// TIA Portal project "modbus-tcp-as-server" (V17)

(* hardware
DEVICE "S7-1200 station_1"  S7-1200 Station
   slot 0: "Rack_0"  S7-1200 Rack  Rack  V1.0
   slot 1: "PLC_1"  CPU 1214C DC/DC/DC  6ES7 214-1AG40-0XB0  V4.5
   slot 101: "CM 1241 (RS422/485)_1"  6ES7 241-1CH32-0XB0  V2.2
*)

// ===== PLC "PLC_1"  CPU 1214C DC/DC/DC =====

VAR_GLOBAL   // PLC tag table "Default tag table"
   "System_Byte" AT %MB1 : Byte;
   "FirstScan" AT %M1.0 : Bool;
   "DiagStatusUpdate" AT %M1.1 : Bool;
   "AlwaysTRUE" AT %M1.2 : Bool;
   "AlwaysFALSE" AT %M1.3 : Bool;
   "Clock_Byte" AT %MB0 : Byte;
   "Clock_10Hz" AT %M0.0 : Bool;
   "Clock_5Hz" AT %M0.1 : Bool;
   "Clock_2.5Hz" AT %M0.2 : Bool;
   "Clock_2Hz" AT %M0.3 : Bool;
   "Clock_1.25Hz" AT %M0.4 : Bool;
   "Clock_1Hz" AT %M0.5 : Bool;
   "Clock_0.625Hz" AT %M0.6 : Bool;
   "Clock_0.5Hz" AT %M0.7 : Bool;
   "Bit1s" AT %M2.0 : Bool;
END_VAR

// folder: Global

DATA_BLOCK "ConfigModel"   // DB1
{ S7_Optimized_Access := 'TRUE' }
VERSION : 0.1
   VAR
      Info : Struct
         ProjectName : String := 'Modbus Tcp As Server';
         Client : String := 'Than Ho';
         Authour : String := 'thanho.dut@gmail.com';
         Tel : String := '0933600195';
         "Version" : String := '2023.05.23.001';
      END_STRUCT;
   END_VAR
BEGIN
END_DATA_BLOCK

DATA_BLOCK "ModbusModel"   // DB3
{ S7_Optimized_Access := 'TRUE' }
VERSION : 0.1
   VAR
      Disconnect : Bool := FALSE;
      NDR : Bool := FALSE;   // Write data completed withou error
      DR : Bool := FALSE;   // Read data completed withou error
      Error : Bool := FALSE;   // Instruction finished with error
      Status : Word := 16#7006;   // Detailed error information
      Connect : TCON_IP_v4;
      HoldingRegisters : Array[0..4999] of Word;   // Data buffer write/read
   END_VAR
BEGIN
   Connect.InterfaceId := 64;
   Connect.ID := 16#0001;
   Connect.RemoteAddress.ADDR[1] := 16#00;
   Connect.RemoteAddress.ADDR[2] := 16#00;
   Connect.RemoteAddress.ADDR[3] := 16#00;
   Connect.RemoteAddress.ADDR[4] := 16#00;
   Connect.LocalPort := 502;
   Connect.ConnectionType := 16#0B;
   Connect.ActiveEstablished := FALSE;
   Connect.RemotePort := 0;
   HoldingRegisters[0] := 16#0000;
   HoldingRegisters[1] := 16#0000;
   HoldingRegisters[2] := 16#0000;
   HoldingRegisters[3] := 16#0000;
   HoldingRegisters[4] := 16#0000;
   HoldingRegisters[5] := 16#0000;
   HoldingRegisters[6] := 16#0000;
   HoldingRegisters[7] := 16#0000;
   HoldingRegisters[8] := 16#0000;
   HoldingRegisters[9] := 16#0000;
   HoldingRegisters[10] := 16#0000;
   HoldingRegisters[11] := 16#0000;
   HoldingRegisters[12] := 16#0000;
   HoldingRegisters[13] := 16#0000;
   HoldingRegisters[14] := 16#0000;
   HoldingRegisters[15] := 16#0000;
   HoldingRegisters[16] := 16#0000;
   HoldingRegisters[17] := 16#0000;
   HoldingRegisters[18] := 16#0000;
   HoldingRegisters[19] := 16#0000;
   HoldingRegisters[20] := 16#0000;
   HoldingRegisters[21] := 16#0000;
   HoldingRegisters[22] := 16#0000;
   HoldingRegisters[23] := 16#0000;
   HoldingRegisters[24] := 16#0000;
   HoldingRegisters[25] := 16#0000;
   HoldingRegisters[26] := 16#0000;
   HoldingRegisters[27] := 16#0000;
   HoldingRegisters[28] := 16#0000;
   HoldingRegisters[29] := 16#0000;
   HoldingRegisters[30] := 16#0000;
   HoldingRegisters[31] := 16#0000;
   HoldingRegisters[32] := 16#0000;
   HoldingRegisters[33] := 16#0000;
   HoldingRegisters[34] := 16#0000;
   HoldingRegisters[35] := 16#0000;
   HoldingRegisters[36] := 16#0000;
   HoldingRegisters[37] := 16#0000;
   HoldingRegisters[38] := 16#0000;
   HoldingRegisters[39] := 16#0000;
   HoldingRegisters[40] := 16#0000;
   HoldingRegisters[41] := 16#0000;
   HoldingRegisters[42] := 16#0000;
   HoldingRegisters[43] := 16#0000;
   HoldingRegisters[44] := 16#0000;
   HoldingRegisters[45] := 16#0000;
   HoldingRegisters[46] := 16#0000;
   HoldingRegisters[47] := 16#0000;
   HoldingRegisters[48] := 16#0000;
   HoldingRegisters[49] := 16#0000;
   HoldingRegisters[50] := 16#0000;
   HoldingRegisters[51] := 16#0000;
   HoldingRegisters[52] := 16#0000;
   HoldingRegisters[53] := 16#0000;
   HoldingRegisters[54] := 16#0000;
   HoldingRegisters[55] := 16#0000;
   HoldingRegisters[56] := 16#0000;
   HoldingRegisters[57] := 16#0000;
   HoldingRegisters[58] := 16#0000;
   HoldingRegisters[59] := 16#0000;
   HoldingRegisters[60] := 16#0000;
   HoldingRegisters[61] := 16#0000;
   HoldingRegisters[62] := 16#0000;
   HoldingRegisters[63] := 16#0000;
   HoldingRegisters[64] := 16#0000;
   HoldingRegisters[65] := 16#0000;
   HoldingRegisters[66] := 16#0000;
   HoldingRegisters[67] := 16#0000;
   HoldingRegisters[68] := 16#0000;
   HoldingRegisters[69] := 16#0000;
   HoldingRegisters[70] := 16#0000;
   HoldingRegisters[71] := 16#0000;
   HoldingRegisters[72] := 16#0000;
   HoldingRegisters[73] := 16#0000;
   HoldingRegisters[74] := 16#0000;
   HoldingRegisters[75] := 16#0000;
   HoldingRegisters[76] := 16#0000;
   HoldingRegisters[77] := 16#0000;
   HoldingRegisters[78] := 16#0000;
   HoldingRegisters[79] := 16#0000;
   HoldingRegisters[80] := 16#0000;
   HoldingRegisters[81] := 16#0000;
   HoldingRegisters[82] := 16#0000;
   HoldingRegisters[83] := 16#0000;
   HoldingRegisters[84] := 16#0000;
   HoldingRegisters[85] := 16#0000;
   HoldingRegisters[86] := 16#0000;
   HoldingRegisters[87] := 16#0000;
   HoldingRegisters[88] := 16#0000;
   HoldingRegisters[89] := 16#0000;
   HoldingRegisters[90] := 16#0000;
   HoldingRegisters[91] := 16#0000;
   HoldingRegisters[92] := 16#0000;
   HoldingRegisters[93] := 16#0000;
   HoldingRegisters[94] := 16#0000;
   HoldingRegisters[95] := 16#0000;
   HoldingRegisters[96] := 16#0000;
   HoldingRegisters[97] := 16#0000;
   HoldingRegisters[98] := 16#0000;
   HoldingRegisters[99] := 16#0000;
   HoldingRegisters[100] := 16#0006;
   HoldingRegisters[101] := 16#0000;
   HoldingRegisters[102] := 16#0000;
   HoldingRegisters[103] := 16#0000;
   HoldingRegisters[104] := 16#0000;
   HoldingRegisters[105] := 16#0000;
   HoldingRegisters[106] := 16#0000;
   HoldingRegisters[107] := 16#0000;
   HoldingRegisters[108] := 16#0000;
   HoldingRegisters[109] := 16#0000;
   HoldingRegisters[110] := 16#0000;
   HoldingRegisters[111] := 16#0000;
   HoldingRegisters[112] := 16#0000;
   HoldingRegisters[113] := 16#0000;
   HoldingRegisters[114] := 16#0000;
   HoldingRegisters[115] := 16#0000;
   HoldingRegisters[116] := 16#0000;
   HoldingRegisters[117] := 16#0000;
   HoldingRegisters[118] := 16#0000;
   HoldingRegisters[119] := 16#0000;
   HoldingRegisters[120] := 16#0000;
   HoldingRegisters[121] := 16#0000;
   HoldingRegisters[122] := 16#0000;
   HoldingRegisters[123] := 16#0000;
   HoldingRegisters[124] := 16#0000;
   HoldingRegisters[125] := 16#0000;
   HoldingRegisters[126] := 16#0000;
   HoldingRegisters[127] := 16#0000;
   HoldingRegisters[128] := 16#0000;
   HoldingRegisters[129] := 16#0000;
   HoldingRegisters[130] := 16#0000;
   HoldingRegisters[131] := 16#0000;
   HoldingRegisters[132] := 16#0000;
   HoldingRegisters[133] := 16#0000;
   HoldingRegisters[134] := 16#0000;
   HoldingRegisters[135] := 16#0000;
   HoldingRegisters[136] := 16#0000;
   HoldingRegisters[137] := 16#0000;
   HoldingRegisters[138] := 16#0000;
   HoldingRegisters[139] := 16#0000;
   HoldingRegisters[140] := 16#0000;
   HoldingRegisters[141] := 16#0000;
   HoldingRegisters[142] := 16#0000;
   HoldingRegisters[143] := 16#0000;
   HoldingRegisters[144] := 16#0000;
   HoldingRegisters[145] := 16#0000;
   HoldingRegisters[146] := 16#0000;
   HoldingRegisters[147] := 16#0000;
   HoldingRegisters[148] := 16#0000;
   HoldingRegisters[149] := 16#0000;
   HoldingRegisters[150] := 16#0000;
   HoldingRegisters[151] := 16#0000;
   HoldingRegisters[152] := 16#0000;
   HoldingRegisters[153] := 16#0000;
   HoldingRegisters[154] := 16#0000;
   HoldingRegisters[155] := 16#0000;
   HoldingRegisters[156] := 16#0000;
   HoldingRegisters[157] := 16#0000;
   HoldingRegisters[158] := 16#0000;
   HoldingRegisters[159] := 16#0000;
   HoldingRegisters[160] := 16#0000;
   HoldingRegisters[161] := 16#0000;
   HoldingRegisters[162] := 16#0000;
   HoldingRegisters[163] := 16#0000;
   HoldingRegisters[164] := 16#0000;
   HoldingRegisters[165] := 16#0000;
   HoldingRegisters[166] := 16#0000;
   HoldingRegisters[167] := 16#0000;
   HoldingRegisters[168] := 16#0000;
   HoldingRegisters[169] := 16#0000;
   HoldingRegisters[170] := 16#0000;
   HoldingRegisters[171] := 16#0000;
   HoldingRegisters[172] := 16#0000;
   HoldingRegisters[173] := 16#0000;
   HoldingRegisters[174] := 16#0000;
   HoldingRegisters[175] := 16#0000;
   HoldingRegisters[176] := 16#0000;
   HoldingRegisters[177] := 16#0000;
   HoldingRegisters[178] := 16#0000;
   HoldingRegisters[179] := 16#0000;
   HoldingRegisters[180] := 16#0000;
   HoldingRegisters[181] := 16#0000;
   HoldingRegisters[182] := 16#0000;
   HoldingRegisters[183] := 16#0000;
   HoldingRegisters[184] := 16#0000;
   HoldingRegisters[185] := 16#0000;
   HoldingRegisters[186] := 16#0000;
   HoldingRegisters[187] := 16#0000;
   HoldingRegisters[188] := 16#0000;
   HoldingRegisters[189] := 16#0000;
   HoldingRegisters[190] := 16#0000;
   HoldingRegisters[191] := 16#0000;
   HoldingRegisters[192] := 16#0000;
   HoldingRegisters[193] := 16#0000;
   HoldingRegisters[194] := 16#0000;
   HoldingRegisters[195] := 16#0000;
   HoldingRegisters[196] := 16#0000;
   HoldingRegisters[197] := 16#0000;
   HoldingRegisters[198] := 16#0000;
   HoldingRegisters[199] := 16#0000;
   HoldingRegisters[200] := 16#0000;
   HoldingRegisters[201] := 16#0000;
   HoldingRegisters[202] := 16#0000;
   HoldingRegisters[203] := 16#0000;
   HoldingRegisters[204] := 16#0000;
   HoldingRegisters[205] := 16#0000;
   HoldingRegisters[206] := 16#0000;
   HoldingRegisters[207] := 16#0000;
   HoldingRegisters[208] := 16#0000;
   HoldingRegisters[209] := 16#0000;
   HoldingRegisters[210] := 16#0000;
   HoldingRegisters[211] := 16#0000;
   HoldingRegisters[212] := 16#0000;
   HoldingRegisters[213] := 16#0000;
   HoldingRegisters[214] := 16#0000;
   HoldingRegisters[215] := 16#0000;
   HoldingRegisters[216] := 16#0000;
   HoldingRegisters[217] := 16#0000;
   HoldingRegisters[218] := 16#0000;
   HoldingRegisters[219] := 16#0000;
   HoldingRegisters[220] := 16#0000;
   HoldingRegisters[221] := 16#0000;
   HoldingRegisters[222] := 16#0000;
   HoldingRegisters[223] := 16#0000;
   HoldingRegisters[224] := 16#0000;
   HoldingRegisters[225] := 16#0000;
   HoldingRegisters[226] := 16#0000;
   HoldingRegisters[227] := 16#0000;
   HoldingRegisters[228] := 16#0000;
   HoldingRegisters[229] := 16#0000;
   HoldingRegisters[230] := 16#0000;
   HoldingRegisters[231] := 16#0000;
   HoldingRegisters[232] := 16#0000;
   HoldingRegisters[233] := 16#0000;
   HoldingRegisters[234] := 16#0000;
   HoldingRegisters[235] := 16#0000;
   HoldingRegisters[236] := 16#0000;
   HoldingRegisters[237] := 16#0000;
   HoldingRegisters[238] := 16#0000;
   HoldingRegisters[239] := 16#0000;
   HoldingRegisters[240] := 16#0000;
   HoldingRegisters[241] := 16#0000;
   HoldingRegisters[242] := 16#0000;
   HoldingRegisters[243] := 16#0000;
   HoldingRegisters[244] := 16#0000;
   HoldingRegisters[245] := 16#0000;
   HoldingRegisters[246] := 16#0000;
   HoldingRegisters[247] := 16#0000;
   HoldingRegisters[248] := 16#0000;
   HoldingRegisters[249] := 16#0000;
   HoldingRegisters[250] := 16#0000;
   HoldingRegisters[251] := 16#0000;
   HoldingRegisters[252] := 16#0000;
   HoldingRegisters[253] := 16#0000;
   HoldingRegisters[254] := 16#0000;
   HoldingRegisters[255] := 16#0000;
   HoldingRegisters[256] := 16#0000;
   HoldingRegisters[257] := 16#0000;
   HoldingRegisters[258] := 16#0000;
   HoldingRegisters[259] := 16#0000;
   HoldingRegisters[260] := 16#0000;
   HoldingRegisters[261] := 16#0000;
   HoldingRegisters[262] := 16#0000;
   HoldingRegisters[263] := 16#0000;
   HoldingRegisters[264] := 16#0000;
   HoldingRegisters[265] := 16#0000;
   HoldingRegisters[266] := 16#0000;
   HoldingRegisters[267] := 16#0000;
   HoldingRegisters[268] := 16#0000;
   HoldingRegisters[269] := 16#0000;
   HoldingRegisters[270] := 16#0000;
   HoldingRegisters[271] := 16#0000;
   HoldingRegisters[272] := 16#0000;
   HoldingRegisters[273] := 16#0000;
   HoldingRegisters[274] := 16#0000;
   HoldingRegisters[275] := 16#0000;
   HoldingRegisters[276] := 16#0000;
   HoldingRegisters[277] := 16#0000;
   HoldingRegisters[278] := 16#0000;
   HoldingRegisters[279] := 16#0000;
   HoldingRegisters[280] := 16#0000;
   HoldingRegisters[281] := 16#0000;
   HoldingRegisters[282] := 16#0000;
   HoldingRegisters[283] := 16#0000;
   HoldingRegisters[284] := 16#0000;
   HoldingRegisters[285] := 16#0000;
   HoldingRegisters[286] := 16#0000;
   HoldingRegisters[287] := 16#0000;
   HoldingRegisters[288] := 16#0000;
   HoldingRegisters[289] := 16#0000;
   HoldingRegisters[290] := 16#0000;
   HoldingRegisters[291] := 16#0000;
   HoldingRegisters[292] := 16#0000;
   HoldingRegisters[293] := 16#0000;
   HoldingRegisters[294] := 16#0000;
   HoldingRegisters[295] := 16#0000;
   HoldingRegisters[296] := 16#0000;
   HoldingRegisters[297] := 16#0000;
   HoldingRegisters[298] := 16#0000;
   HoldingRegisters[299] := 16#0000;
   HoldingRegisters[300] := 16#0000;
   HoldingRegisters[301] := 16#0000;
   HoldingRegisters[302] := 16#0000;
   HoldingRegisters[303] := 16#0000;
   HoldingRegisters[304] := 16#0000;
   HoldingRegisters[305] := 16#0000;
   HoldingRegisters[306] := 16#0000;
   HoldingRegisters[307] := 16#0000;
   HoldingRegisters[308] := 16#0000;
   HoldingRegisters[309] := 16#0000;
   HoldingRegisters[310] := 16#0000;
   HoldingRegisters[311] := 16#0000;
   HoldingRegisters[312] := 16#0000;
   HoldingRegisters[313] := 16#0000;
   HoldingRegisters[314] := 16#0000;
   HoldingRegisters[315] := 16#0000;
   HoldingRegisters[316] := 16#0000;
   HoldingRegisters[317] := 16#0000;
   HoldingRegisters[318] := 16#0000;
   HoldingRegisters[319] := 16#0000;
   HoldingRegisters[320] := 16#0000;
   HoldingRegisters[321] := 16#0000;
   HoldingRegisters[322] := 16#0000;
   HoldingRegisters[323] := 16#0000;
   HoldingRegisters[324] := 16#0000;
   HoldingRegisters[325] := 16#0000;
   HoldingRegisters[326] := 16#0000;
   HoldingRegisters[327] := 16#0000;
   HoldingRegisters[328] := 16#0000;
   HoldingRegisters[329] := 16#0000;
   HoldingRegisters[330] := 16#0000;
   HoldingRegisters[331] := 16#0000;
   HoldingRegisters[332] := 16#0000;
   HoldingRegisters[333] := 16#0000;
   HoldingRegisters[334] := 16#0000;
   HoldingRegisters[335] := 16#0000;
   HoldingRegisters[336] := 16#0000;
   HoldingRegisters[337] := 16#0000;
   HoldingRegisters[338] := 16#0000;
   HoldingRegisters[339] := 16#0000;
   HoldingRegisters[340] := 16#0000;
   HoldingRegisters[341] := 16#0000;
   HoldingRegisters[342] := 16#0000;
   HoldingRegisters[343] := 16#0000;
   HoldingRegisters[344] := 16#0000;
   HoldingRegisters[345] := 16#0000;
   HoldingRegisters[346] := 16#0000;
   HoldingRegisters[347] := 16#0000;
   HoldingRegisters[348] := 16#0000;
   HoldingRegisters[349] := 16#0000;
   HoldingRegisters[350] := 16#0000;
   HoldingRegisters[351] := 16#0000;
   HoldingRegisters[352] := 16#0000;
   HoldingRegisters[353] := 16#0000;
   HoldingRegisters[354] := 16#0000;
   HoldingRegisters[355] := 16#0000;
   HoldingRegisters[356] := 16#0000;
   HoldingRegisters[357] := 16#0000;
   HoldingRegisters[358] := 16#0000;
   HoldingRegisters[359] := 16#0000;
   HoldingRegisters[360] := 16#0000;
   HoldingRegisters[361] := 16#0000;
   HoldingRegisters[362] := 16#0000;
   HoldingRegisters[363] := 16#0000;
   HoldingRegisters[364] := 16#0000;
   HoldingRegisters[365] := 16#0000;
   HoldingRegisters[366] := 16#0000;
   HoldingRegisters[367] := 16#0000;
   HoldingRegisters[368] := 16#0000;
   HoldingRegisters[369] := 16#0000;
   HoldingRegisters[370] := 16#0000;
   HoldingRegisters[371] := 16#0000;
   HoldingRegisters[372] := 16#0000;
   HoldingRegisters[373] := 16#0000;
   HoldingRegisters[374] := 16#0000;
   HoldingRegisters[375] := 16#0000;
   HoldingRegisters[376] := 16#0000;
   HoldingRegisters[377] := 16#0000;
   HoldingRegisters[378] := 16#0000;
   HoldingRegisters[379] := 16#0000;
   HoldingRegisters[380] := 16#0000;
   HoldingRegisters[381] := 16#0000;
   HoldingRegisters[382] := 16#0000;
   HoldingRegisters[383] := 16#0000;
   HoldingRegisters[384] := 16#0000;
   HoldingRegisters[385] := 16#0000;
   HoldingRegisters[386] := 16#0000;
   HoldingRegisters[387] := 16#0000;
   HoldingRegisters[388] := 16#0000;
   HoldingRegisters[389] := 16#0000;
   HoldingRegisters[390] := 16#0000;
   HoldingRegisters[391] := 16#0000;
   HoldingRegisters[392] := 16#0000;
   HoldingRegisters[393] := 16#0000;
   HoldingRegisters[394] := 16#0000;
   HoldingRegisters[395] := 16#0000;
   HoldingRegisters[396] := 16#0000;
   HoldingRegisters[397] := 16#0000;
   HoldingRegisters[398] := 16#0000;
   HoldingRegisters[399] := 16#0000;
   HoldingRegisters[400] := 16#0000;
   HoldingRegisters[401] := 16#0000;
   HoldingRegisters[402] := 16#0000;
   HoldingRegisters[403] := 16#0000;
   HoldingRegisters[404] := 16#0000;
   HoldingRegisters[405] := 16#0000;
   HoldingRegisters[406] := 16#0000;
   HoldingRegisters[407] := 16#0000;
   HoldingRegisters[408] := 16#0000;
   HoldingRegisters[409] := 16#0000;
   HoldingRegisters[410] := 16#0000;
   HoldingRegisters[411] := 16#0000;
   HoldingRegisters[412] := 16#0000;
   HoldingRegisters[413] := 16#0000;
   HoldingRegisters[414] := 16#0000;
   HoldingRegisters[415] := 16#0000;
   HoldingRegisters[416] := 16#0000;
   HoldingRegisters[417] := 16#0000;
   HoldingRegisters[418] := 16#0000;
   HoldingRegisters[419] := 16#0000;
   HoldingRegisters[420] := 16#0000;
   HoldingRegisters[421] := 16#0000;
   HoldingRegisters[422] := 16#0000;
   HoldingRegisters[423] := 16#0000;
   HoldingRegisters[424] := 16#0000;
   HoldingRegisters[425] := 16#0000;
   HoldingRegisters[426] := 16#0000;
   HoldingRegisters[427] := 16#0000;
   HoldingRegisters[428] := 16#0000;
   HoldingRegisters[429] := 16#0000;
   HoldingRegisters[430] := 16#0000;
   HoldingRegisters[431] := 16#0000;
   HoldingRegisters[432] := 16#0000;
   HoldingRegisters[433] := 16#0000;
   HoldingRegisters[434] := 16#0000;
   HoldingRegisters[435] := 16#0000;
   HoldingRegisters[436] := 16#0000;
   HoldingRegisters[437] := 16#0000;
   HoldingRegisters[438] := 16#0000;
   HoldingRegisters[439] := 16#0000;
   HoldingRegisters[440] := 16#0000;
   HoldingRegisters[441] := 16#0000;
   HoldingRegisters[442] := 16#0000;
   HoldingRegisters[443] := 16#0000;
   HoldingRegisters[444] := 16#0000;
   HoldingRegisters[445] := 16#0000;
   HoldingRegisters[446] := 16#0000;
   HoldingRegisters[447] := 16#0000;
   HoldingRegisters[448] := 16#0000;
   HoldingRegisters[449] := 16#0000;
   HoldingRegisters[450] := 16#0000;
   HoldingRegisters[451] := 16#0000;
   HoldingRegisters[452] := 16#0000;
   HoldingRegisters[453] := 16#0000;
   HoldingRegisters[454] := 16#0000;
   HoldingRegisters[455] := 16#0000;
   HoldingRegisters[456] := 16#0000;
   HoldingRegisters[457] := 16#0000;
   HoldingRegisters[458] := 16#0000;
   HoldingRegisters[459] := 16#0000;
   HoldingRegisters[460] := 16#0000;
   HoldingRegisters[461] := 16#0000;
   HoldingRegisters[462] := 16#0000;
   HoldingRegisters[463] := 16#0000;
   HoldingRegisters[464] := 16#0000;
   HoldingRegisters[465] := 16#0000;
   HoldingRegisters[466] := 16#0000;
   HoldingRegisters[467] := 16#0000;
   HoldingRegisters[468] := 16#0000;
   HoldingRegisters[469] := 16#0000;
   HoldingRegisters[470] := 16#0000;
   HoldingRegisters[471] := 16#0000;
   HoldingRegisters[472] := 16#0000;
   HoldingRegisters[473] := 16#0000;
   HoldingRegisters[474] := 16#0000;
   HoldingRegisters[475] := 16#0000;
   HoldingRegisters[476] := 16#0000;
   HoldingRegisters[477] := 16#0000;
   HoldingRegisters[478] := 16#0000;
   HoldingRegisters[479] := 16#0000;
   HoldingRegisters[480] := 16#0000;
   HoldingRegisters[481] := 16#0000;
   HoldingRegisters[482] := 16#0000;
   HoldingRegisters[483] := 16#0000;
   HoldingRegisters[484] := 16#0000;
   HoldingRegisters[485] := 16#0000;
   HoldingRegisters[486] := 16#0000;
   HoldingRegisters[487] := 16#0000;
   HoldingRegisters[488] := 16#0000;
   HoldingRegisters[489] := 16#0000;
   HoldingRegisters[490] := 16#0000;
   HoldingRegisters[491] := 16#0000;
   HoldingRegisters[492] := 16#0000;
   HoldingRegisters[493] := 16#0000;
   HoldingRegisters[494] := 16#0000;
   HoldingRegisters[495] := 16#0000;
   HoldingRegisters[496] := 16#0000;
   HoldingRegisters[497] := 16#0000;
   HoldingRegisters[498] := 16#0000;
   HoldingRegisters[499] := 16#0000;
   HoldingRegisters[500] := 16#0000;
   HoldingRegisters[501] := 16#0000;
   HoldingRegisters[502] := 16#0000;
   HoldingRegisters[503] := 16#0000;
   HoldingRegisters[504] := 16#0000;
   HoldingRegisters[505] := 16#0000;
   HoldingRegisters[506] := 16#0000;
   HoldingRegisters[507] := 16#0000;
   HoldingRegisters[508] := 16#0000;
   HoldingRegisters[509] := 16#0000;
   HoldingRegisters[510] := 16#0000;
   HoldingRegisters[511] := 16#0000;
   HoldingRegisters[512] := 16#0000;
   HoldingRegisters[513] := 16#0000;
   HoldingRegisters[514] := 16#0000;
   HoldingRegisters[515] := 16#0000;
   HoldingRegisters[516] := 16#0000;
   HoldingRegisters[517] := 16#0000;
   HoldingRegisters[518] := 16#0000;
   HoldingRegisters[519] := 16#0000;
   HoldingRegisters[520] := 16#0000;
   HoldingRegisters[521] := 16#0000;
   HoldingRegisters[522] := 16#0000;
   HoldingRegisters[523] := 16#0000;
   HoldingRegisters[524] := 16#0000;
   HoldingRegisters[525] := 16#0000;
   HoldingRegisters[526] := 16#0000;
   HoldingRegisters[527] := 16#0000;
   HoldingRegisters[528] := 16#0000;
   HoldingRegisters[529] := 16#0000;
   HoldingRegisters[530] := 16#0000;
   HoldingRegisters[531] := 16#0000;
   HoldingRegisters[532] := 16#0000;
   HoldingRegisters[533] := 16#0000;
   HoldingRegisters[534] := 16#0000;
   HoldingRegisters[535] := 16#0000;
   HoldingRegisters[536] := 16#0000;
   HoldingRegisters[537] := 16#0000;
   HoldingRegisters[538] := 16#0000;
   HoldingRegisters[539] := 16#0000;
   HoldingRegisters[540] := 16#0000;
   HoldingRegisters[541] := 16#0000;
   HoldingRegisters[542] := 16#0000;
   HoldingRegisters[543] := 16#0000;
   HoldingRegisters[544] := 16#0000;
   HoldingRegisters[545] := 16#0000;
   HoldingRegisters[546] := 16#0000;
   HoldingRegisters[547] := 16#0000;
   HoldingRegisters[548] := 16#0000;
   HoldingRegisters[549] := 16#0000;
   HoldingRegisters[550] := 16#0000;
   HoldingRegisters[551] := 16#0000;
   HoldingRegisters[552] := 16#0000;
   HoldingRegisters[553] := 16#0000;
   HoldingRegisters[554] := 16#0000;
   HoldingRegisters[555] := 16#0000;
   HoldingRegisters[556] := 16#0000;
   HoldingRegisters[557] := 16#0000;
   HoldingRegisters[558] := 16#0000;
   HoldingRegisters[559] := 16#0000;
   HoldingRegisters[560] := 16#0000;
   HoldingRegisters[561] := 16#0000;
   HoldingRegisters[562] := 16#0000;
   HoldingRegisters[563] := 16#0000;
   HoldingRegisters[564] := 16#0000;
   HoldingRegisters[565] := 16#0000;
   HoldingRegisters[566] := 16#0000;
   HoldingRegisters[567] := 16#0000;
   HoldingRegisters[568] := 16#0000;
   HoldingRegisters[569] := 16#0000;
   HoldingRegisters[570] := 16#0000;
   HoldingRegisters[571] := 16#0000;
   HoldingRegisters[572] := 16#0000;
   HoldingRegisters[573] := 16#0000;
   HoldingRegisters[574] := 16#0000;
   HoldingRegisters[575] := 16#0000;
   HoldingRegisters[576] := 16#0000;
   HoldingRegisters[577] := 16#0000;
   HoldingRegisters[578] := 16#0000;
   HoldingRegisters[579] := 16#0000;
   HoldingRegisters[580] := 16#0000;
   HoldingRegisters[581] := 16#0000;
   HoldingRegisters[582] := 16#0000;
   HoldingRegisters[583] := 16#0000;
   HoldingRegisters[584] := 16#0000;
   HoldingRegisters[585] := 16#0000;
   HoldingRegisters[586] := 16#0000;
   HoldingRegisters[587] := 16#0000;
   HoldingRegisters[588] := 16#0000;
   HoldingRegisters[589] := 16#0000;
   HoldingRegisters[590] := 16#0000;
   HoldingRegisters[591] := 16#0000;
   HoldingRegisters[592] := 16#0000;
   HoldingRegisters[593] := 16#0000;
   HoldingRegisters[594] := 16#0000;
   HoldingRegisters[595] := 16#0000;
   HoldingRegisters[596] := 16#0000;
   HoldingRegisters[597] := 16#0000;
   HoldingRegisters[598] := 16#0000;
   HoldingRegisters[599] := 16#0000;
   HoldingRegisters[600] := 16#0000;
   HoldingRegisters[601] := 16#0000;
   HoldingRegisters[602] := 16#0000;
   HoldingRegisters[603] := 16#0000;
   HoldingRegisters[604] := 16#0000;
   HoldingRegisters[605] := 16#0000;
   HoldingRegisters[606] := 16#0000;
   HoldingRegisters[607] := 16#0000;
   HoldingRegisters[608] := 16#0000;
   HoldingRegisters[609] := 16#0000;
   HoldingRegisters[610] := 16#0000;
   HoldingRegisters[611] := 16#0000;
   HoldingRegisters[612] := 16#0000;
   HoldingRegisters[613] := 16#0000;
   HoldingRegisters[614] := 16#0000;
   HoldingRegisters[615] := 16#0000;
   HoldingRegisters[616] := 16#0000;
   HoldingRegisters[617] := 16#0000;
   HoldingRegisters[618] := 16#0000;
   HoldingRegisters[619] := 16#0000;
   HoldingRegisters[620] := 16#0000;
   HoldingRegisters[621] := 16#0000;
   HoldingRegisters[622] := 16#0000;
   HoldingRegisters[623] := 16#0000;
   HoldingRegisters[624] := 16#0000;
   HoldingRegisters[625] := 16#0000;
   HoldingRegisters[626] := 16#0000;
   HoldingRegisters[627] := 16#0000;
   HoldingRegisters[628] := 16#0000;
   HoldingRegisters[629] := 16#0000;
   HoldingRegisters[630] := 16#0000;
   HoldingRegisters[631] := 16#0000;
   HoldingRegisters[632] := 16#0000;
   HoldingRegisters[633] := 16#0000;
   HoldingRegisters[634] := 16#0000;
   HoldingRegisters[635] := 16#0000;
   HoldingRegisters[636] := 16#0000;
   HoldingRegisters[637] := 16#0000;
   HoldingRegisters[638] := 16#0000;
   HoldingRegisters[639] := 16#0000;
   HoldingRegisters[640] := 16#0000;
   HoldingRegisters[641] := 16#0000;
   HoldingRegisters[642] := 16#0000;
   HoldingRegisters[643] := 16#0000;
   HoldingRegisters[644] := 16#0000;
   HoldingRegisters[645] := 16#0000;
   HoldingRegisters[646] := 16#0000;
   HoldingRegisters[647] := 16#0000;
   HoldingRegisters[648] := 16#0000;
   HoldingRegisters[649] := 16#0000;
   HoldingRegisters[650] := 16#0000;
   HoldingRegisters[651] := 16#0000;
   HoldingRegisters[652] := 16#0000;
   HoldingRegisters[653] := 16#0000;
   HoldingRegisters[654] := 16#0000;
   HoldingRegisters[655] := 16#0000;
   HoldingRegisters[656] := 16#0000;
   HoldingRegisters[657] := 16#0000;
   HoldingRegisters[658] := 16#0000;
   HoldingRegisters[659] := 16#0000;
   HoldingRegisters[660] := 16#0000;
   HoldingRegisters[661] := 16#0000;
   HoldingRegisters[662] := 16#0000;
   HoldingRegisters[663] := 16#0000;
   HoldingRegisters[664] := 16#0000;
   HoldingRegisters[665] := 16#0000;
   HoldingRegisters[666] := 16#0000;
   HoldingRegisters[667] := 16#0000;
   HoldingRegisters[668] := 16#0000;
   HoldingRegisters[669] := 16#0000;
   HoldingRegisters[670] := 16#0000;
   HoldingRegisters[671] := 16#0000;
   HoldingRegisters[672] := 16#0000;
   HoldingRegisters[673] := 16#0000;
   HoldingRegisters[674] := 16#0000;
   HoldingRegisters[675] := 16#0000;
   HoldingRegisters[676] := 16#0000;
   HoldingRegisters[677] := 16#0000;
   HoldingRegisters[678] := 16#0000;
   HoldingRegisters[679] := 16#0000;
   HoldingRegisters[680] := 16#0000;
   HoldingRegisters[681] := 16#0000;
   HoldingRegisters[682] := 16#0000;
   HoldingRegisters[683] := 16#0000;
   HoldingRegisters[684] := 16#0000;
   HoldingRegisters[685] := 16#0000;
   HoldingRegisters[686] := 16#0000;
   HoldingRegisters[687] := 16#0000;
   HoldingRegisters[688] := 16#0000;
   HoldingRegisters[689] := 16#0000;
   HoldingRegisters[690] := 16#0000;
   HoldingRegisters[691] := 16#0000;
   HoldingRegisters[692] := 16#0000;
   HoldingRegisters[693] := 16#0000;
   HoldingRegisters[694] := 16#0000;
   HoldingRegisters[695] := 16#0000;
   HoldingRegisters[696] := 16#0000;
   HoldingRegisters[697] := 16#0000;
   HoldingRegisters[698] := 16#0000;
   HoldingRegisters[699] := 16#0000;
   HoldingRegisters[700] := 16#0000;
   HoldingRegisters[701] := 16#0000;
   HoldingRegisters[702] := 16#0000;
   HoldingRegisters[703] := 16#0000;
   HoldingRegisters[704] := 16#0000;
   HoldingRegisters[705] := 16#0000;
   HoldingRegisters[706] := 16#0000;
   HoldingRegisters[707] := 16#0000;
   HoldingRegisters[708] := 16#0000;
   HoldingRegisters[709] := 16#0000;
   HoldingRegisters[710] := 16#0000;
   HoldingRegisters[711] := 16#0000;
   HoldingRegisters[712] := 16#0000;
   HoldingRegisters[713] := 16#0000;
   HoldingRegisters[714] := 16#0000;
   HoldingRegisters[715] := 16#0000;
   HoldingRegisters[716] := 16#0000;
   HoldingRegisters[717] := 16#0000;
   HoldingRegisters[718] := 16#0000;
   HoldingRegisters[719] := 16#0000;
   HoldingRegisters[720] := 16#0000;
   HoldingRegisters[721] := 16#0000;
   HoldingRegisters[722] := 16#0000;
   HoldingRegisters[723] := 16#0000;
   HoldingRegisters[724] := 16#0000;
   HoldingRegisters[725] := 16#0000;
   HoldingRegisters[726] := 16#0000;
   HoldingRegisters[727] := 16#0000;
   HoldingRegisters[728] := 16#0000;
   HoldingRegisters[729] := 16#0000;
   HoldingRegisters[730] := 16#0000;
   HoldingRegisters[731] := 16#0000;
   HoldingRegisters[732] := 16#0000;
   HoldingRegisters[733] := 16#0000;
   HoldingRegisters[734] := 16#0000;
   HoldingRegisters[735] := 16#0000;
   HoldingRegisters[736] := 16#0000;
   HoldingRegisters[737] := 16#0000;
   HoldingRegisters[738] := 16#0000;
   HoldingRegisters[739] := 16#0000;
   HoldingRegisters[740] := 16#0000;
   HoldingRegisters[741] := 16#0000;
   HoldingRegisters[742] := 16#0000;
   HoldingRegisters[743] := 16#0000;
   HoldingRegisters[744] := 16#0000;
   HoldingRegisters[745] := 16#0000;
   HoldingRegisters[746] := 16#0000;
   HoldingRegisters[747] := 16#0000;
   HoldingRegisters[748] := 16#0000;
   HoldingRegisters[749] := 16#0000;
   HoldingRegisters[750] := 16#0000;
   HoldingRegisters[751] := 16#0000;
   HoldingRegisters[752] := 16#0000;
   HoldingRegisters[753] := 16#0000;
   HoldingRegisters[754] := 16#0000;
   HoldingRegisters[755] := 16#0000;
   HoldingRegisters[756] := 16#0000;
   HoldingRegisters[757] := 16#0000;
   HoldingRegisters[758] := 16#0000;
   HoldingRegisters[759] := 16#0000;
   HoldingRegisters[760] := 16#0000;
   HoldingRegisters[761] := 16#0000;
   HoldingRegisters[762] := 16#0000;
   HoldingRegisters[763] := 16#0000;
   HoldingRegisters[764] := 16#0000;
   HoldingRegisters[765] := 16#0000;
   HoldingRegisters[766] := 16#0000;
   HoldingRegisters[767] := 16#0000;
   HoldingRegisters[768] := 16#0000;
   HoldingRegisters[769] := 16#0000;
   HoldingRegisters[770] := 16#0000;
   HoldingRegisters[771] := 16#0000;
   HoldingRegisters[772] := 16#0000;
   HoldingRegisters[773] := 16#0000;
   HoldingRegisters[774] := 16#0000;
   HoldingRegisters[775] := 16#0000;
   HoldingRegisters[776] := 16#0000;
   HoldingRegisters[777] := 16#0000;
   HoldingRegisters[778] := 16#0000;
   HoldingRegisters[779] := 16#0000;
   HoldingRegisters[780] := 16#0000;
   HoldingRegisters[781] := 16#0000;
   HoldingRegisters[782] := 16#0000;
   HoldingRegisters[783] := 16#0000;
   HoldingRegisters[784] := 16#0000;
   HoldingRegisters[785] := 16#0000;
   HoldingRegisters[786] := 16#0000;
   HoldingRegisters[787] := 16#0000;
   HoldingRegisters[788] := 16#0000;
   HoldingRegisters[789] := 16#0000;
   HoldingRegisters[790] := 16#0000;
   HoldingRegisters[791] := 16#0000;
   HoldingRegisters[792] := 16#0000;
   HoldingRegisters[793] := 16#0000;
   HoldingRegisters[794] := 16#0000;
   HoldingRegisters[795] := 16#0000;
   HoldingRegisters[796] := 16#0000;
   HoldingRegisters[797] := 16#0000;
   HoldingRegisters[798] := 16#0000;
   HoldingRegisters[799] := 16#0000;
   HoldingRegisters[800] := 16#0000;
   HoldingRegisters[801] := 16#0000;
   HoldingRegisters[802] := 16#0000;
   HoldingRegisters[803] := 16#0000;
   HoldingRegisters[804] := 16#0000;
   HoldingRegisters[805] := 16#0000;
   HoldingRegisters[806] := 16#0000;
   HoldingRegisters[807] := 16#0000;
   HoldingRegisters[808] := 16#0000;
   HoldingRegisters[809] := 16#0000;
   HoldingRegisters[810] := 16#0000;
   HoldingRegisters[811] := 16#0000;
   HoldingRegisters[812] := 16#0000;
   HoldingRegisters[813] := 16#0000;
   HoldingRegisters[814] := 16#0000;
   HoldingRegisters[815] := 16#0000;
   HoldingRegisters[816] := 16#0000;
   HoldingRegisters[817] := 16#0000;
   HoldingRegisters[818] := 16#0000;
   HoldingRegisters[819] := 16#0000;
   HoldingRegisters[820] := 16#0000;
   HoldingRegisters[821] := 16#0000;
   HoldingRegisters[822] := 16#0000;
   HoldingRegisters[823] := 16#0000;
   HoldingRegisters[824] := 16#0000;
   HoldingRegisters[825] := 16#0000;
   HoldingRegisters[826] := 16#0000;
   HoldingRegisters[827] := 16#0000;
   HoldingRegisters[828] := 16#0000;
   HoldingRegisters[829] := 16#0000;
   HoldingRegisters[830] := 16#0000;
   HoldingRegisters[831] := 16#0000;
   HoldingRegisters[832] := 16#0000;
   HoldingRegisters[833] := 16#0000;
   HoldingRegisters[834] := 16#0000;
   HoldingRegisters[835] := 16#0000;
   HoldingRegisters[836] := 16#0000;
   HoldingRegisters[837] := 16#0000;
   HoldingRegisters[838] := 16#0000;
   HoldingRegisters[839] := 16#0000;
   HoldingRegisters[840] := 16#0000;
   HoldingRegisters[841] := 16#0000;
   HoldingRegisters[842] := 16#0000;
   HoldingRegisters[843] := 16#0000;
   HoldingRegisters[844] := 16#0000;
   HoldingRegisters[845] := 16#0000;
   HoldingRegisters[846] := 16#0000;
   HoldingRegisters[847] := 16#0000;
   HoldingRegisters[848] := 16#0000;
   HoldingRegisters[849] := 16#0000;
   HoldingRegisters[850] := 16#0000;
   HoldingRegisters[851] := 16#0000;
   HoldingRegisters[852] := 16#0000;
   HoldingRegisters[853] := 16#0000;
   HoldingRegisters[854] := 16#0000;
   HoldingRegisters[855] := 16#0000;
   HoldingRegisters[856] := 16#0000;
   HoldingRegisters[857] := 16#0000;
   HoldingRegisters[858] := 16#0000;
   HoldingRegisters[859] := 16#0000;
   HoldingRegisters[860] := 16#0000;
   HoldingRegisters[861] := 16#0000;
   HoldingRegisters[862] := 16#0000;
   HoldingRegisters[863] := 16#0000;
   HoldingRegisters[864] := 16#0000;
   HoldingRegisters[865] := 16#0000;
   HoldingRegisters[866] := 16#0000;
   HoldingRegisters[867] := 16#0000;
   HoldingRegisters[868] := 16#0000;
   HoldingRegisters[869] := 16#0000;
   HoldingRegisters[870] := 16#0000;
   HoldingRegisters[871] := 16#0000;
   HoldingRegisters[872] := 16#0000;
   HoldingRegisters[873] := 16#0000;
   HoldingRegisters[874] := 16#0000;
   HoldingRegisters[875] := 16#0000;
   HoldingRegisters[876] := 16#0000;
   HoldingRegisters[877] := 16#0000;
   HoldingRegisters[878] := 16#0000;
   HoldingRegisters[879] := 16#0000;
   HoldingRegisters[880] := 16#0000;
   HoldingRegisters[881] := 16#0000;
   HoldingRegisters[882] := 16#0000;
   HoldingRegisters[883] := 16#0000;
   HoldingRegisters[884] := 16#0000;
   HoldingRegisters[885] := 16#0000;
   HoldingRegisters[886] := 16#0000;
   HoldingRegisters[887] := 16#0000;
   HoldingRegisters[888] := 16#0000;
   HoldingRegisters[889] := 16#0000;
   HoldingRegisters[890] := 16#0000;
   HoldingRegisters[891] := 16#0000;
   HoldingRegisters[892] := 16#0000;
   HoldingRegisters[893] := 16#0000;
   HoldingRegisters[894] := 16#0000;
   HoldingRegisters[895] := 16#0000;
   HoldingRegisters[896] := 16#0000;
   HoldingRegisters[897] := 16#0000;
   HoldingRegisters[898] := 16#0000;
   HoldingRegisters[899] := 16#0000;
   HoldingRegisters[900] := 16#0000;
   HoldingRegisters[901] := 16#0000;
   HoldingRegisters[902] := 16#0000;
   HoldingRegisters[903] := 16#0000;
   HoldingRegisters[904] := 16#0000;
   HoldingRegisters[905] := 16#0000;
   HoldingRegisters[906] := 16#0000;
   HoldingRegisters[907] := 16#0000;
   HoldingRegisters[908] := 16#0000;
   HoldingRegisters[909] := 16#0000;
   HoldingRegisters[910] := 16#0000;
   HoldingRegisters[911] := 16#0000;
   HoldingRegisters[912] := 16#0000;
   HoldingRegisters[913] := 16#0000;
   HoldingRegisters[914] := 16#0000;
   HoldingRegisters[915] := 16#0000;
   HoldingRegisters[916] := 16#0000;
   HoldingRegisters[917] := 16#0000;
   HoldingRegisters[918] := 16#0000;
   HoldingRegisters[919] := 16#0000;
   HoldingRegisters[920] := 16#0000;
   HoldingRegisters[921] := 16#0000;
   HoldingRegisters[922] := 16#0000;
   HoldingRegisters[923] := 16#0000;
   HoldingRegisters[924] := 16#0000;
   HoldingRegisters[925] := 16#0000;
   HoldingRegisters[926] := 16#0000;
   HoldingRegisters[927] := 16#0000;
   HoldingRegisters[928] := 16#0000;
   HoldingRegisters[929] := 16#0000;
   HoldingRegisters[930] := 16#0000;
   HoldingRegisters[931] := 16#0000;
   HoldingRegisters[932] := 16#0000;
   HoldingRegisters[933] := 16#0000;
   HoldingRegisters[934] := 16#0000;
   HoldingRegisters[935] := 16#0000;
   HoldingRegisters[936] := 16#0000;
   HoldingRegisters[937] := 16#0000;
   HoldingRegisters[938] := 16#0000;
   HoldingRegisters[939] := 16#0000;
   HoldingRegisters[940] := 16#0000;
   HoldingRegisters[941] := 16#0000;
   HoldingRegisters[942] := 16#0000;
   HoldingRegisters[943] := 16#0000;
   HoldingRegisters[944] := 16#0000;
   HoldingRegisters[945] := 16#0000;
   HoldingRegisters[946] := 16#0000;
   HoldingRegisters[947] := 16#0000;
   HoldingRegisters[948] := 16#0000;
   HoldingRegisters[949] := 16#0000;
   HoldingRegisters[950] := 16#0000;
   HoldingRegisters[951] := 16#0000;
   HoldingRegisters[952] := 16#0000;
   HoldingRegisters[953] := 16#0000;
   HoldingRegisters[954] := 16#0000;
   HoldingRegisters[955] := 16#0000;
   HoldingRegisters[956] := 16#0000;
   HoldingRegisters[957] := 16#0000;
   HoldingRegisters[958] := 16#0000;
   HoldingRegisters[959] := 16#0000;
   HoldingRegisters[960] := 16#0000;
   HoldingRegisters[961] := 16#0000;
   HoldingRegisters[962] := 16#0000;
   HoldingRegisters[963] := 16#0000;
   HoldingRegisters[964] := 16#0000;
   HoldingRegisters[965] := 16#0000;
   HoldingRegisters[966] := 16#0000;
   HoldingRegisters[967] := 16#0000;
   HoldingRegisters[968] := 16#0000;
   HoldingRegisters[969] := 16#0000;
   HoldingRegisters[970] := 16#0000;
   HoldingRegisters[971] := 16#0000;
   HoldingRegisters[972] := 16#0000;
   HoldingRegisters[973] := 16#0000;
   HoldingRegisters[974] := 16#0000;
   HoldingRegisters[975] := 16#0000;
   HoldingRegisters[976] := 16#0000;
   HoldingRegisters[977] := 16#0000;
   HoldingRegisters[978] := 16#0000;
   HoldingRegisters[979] := 16#0000;
   HoldingRegisters[980] := 16#0000;
   HoldingRegisters[981] := 16#0000;
   HoldingRegisters[982] := 16#0000;
   HoldingRegisters[983] := 16#0000;
   HoldingRegisters[984] := 16#0000;
   HoldingRegisters[985] := 16#0000;
   HoldingRegisters[986] := 16#0000;
   HoldingRegisters[987] := 16#0000;
   HoldingRegisters[988] := 16#0000;
   HoldingRegisters[989] := 16#0000;
   HoldingRegisters[990] := 16#0000;
   HoldingRegisters[991] := 16#0000;
   HoldingRegisters[992] := 16#0000;
   HoldingRegisters[993] := 16#0000;
   HoldingRegisters[994] := 16#0000;
   HoldingRegisters[995] := 16#0000;
   HoldingRegisters[996] := 16#0000;
   HoldingRegisters[997] := 16#0000;
   HoldingRegisters[998] := 16#0000;
   HoldingRegisters[999] := 16#0000;
   HoldingRegisters[1000] := 16#0000;
   HoldingRegisters[1001] := 16#0000;
   HoldingRegisters[1002] := 16#0000;
   HoldingRegisters[1003] := 16#0000;
   HoldingRegisters[1004] := 16#0000;
   HoldingRegisters[1005] := 16#0000;
   HoldingRegisters[1006] := 16#0000;
   HoldingRegisters[1007] := 16#0000;
   HoldingRegisters[1008] := 16#0000;
   HoldingRegisters[1009] := 16#0000;
   HoldingRegisters[1010] := 16#0000;
   HoldingRegisters[1011] := 16#0000;
   HoldingRegisters[1012] := 16#0000;
   HoldingRegisters[1013] := 16#0000;
   HoldingRegisters[1014] := 16#0000;
   HoldingRegisters[1015] := 16#0000;
   HoldingRegisters[1016] := 16#0000;
   HoldingRegisters[1017] := 16#0000;
   HoldingRegisters[1018] := 16#0000;
   HoldingRegisters[1019] := 16#0000;
   HoldingRegisters[1020] := 16#0000;
   HoldingRegisters[1021] := 16#0000;
   HoldingRegisters[1022] := 16#0000;
   HoldingRegisters[1023] := 16#0000;
   HoldingRegisters[1024] := 16#0000;
   HoldingRegisters[1025] := 16#0000;
   HoldingRegisters[1026] := 16#0000;
   HoldingRegisters[1027] := 16#0000;
   HoldingRegisters[1028] := 16#0000;
   HoldingRegisters[1029] := 16#0000;
   HoldingRegisters[1030] := 16#0000;
   HoldingRegisters[1031] := 16#0000;
   HoldingRegisters[1032] := 16#0000;
   HoldingRegisters[1033] := 16#0000;
   HoldingRegisters[1034] := 16#0000;
   HoldingRegisters[1035] := 16#0000;
   HoldingRegisters[1036] := 16#0000;
   HoldingRegisters[1037] := 16#0000;
   HoldingRegisters[1038] := 16#0000;
   HoldingRegisters[1039] := 16#0000;
   HoldingRegisters[1040] := 16#0000;
   HoldingRegisters[1041] := 16#0000;
   HoldingRegisters[1042] := 16#0000;
   HoldingRegisters[1043] := 16#0000;
   HoldingRegisters[1044] := 16#0000;
   HoldingRegisters[1045] := 16#0000;
   HoldingRegisters[1046] := 16#0000;
   HoldingRegisters[1047] := 16#0000;
   HoldingRegisters[1048] := 16#0000;
   HoldingRegisters[1049] := 16#0000;
   HoldingRegisters[1050] := 16#0000;
   HoldingRegisters[1051] := 16#0000;
   HoldingRegisters[1052] := 16#0000;
   HoldingRegisters[1053] := 16#0000;
   HoldingRegisters[1054] := 16#0000;
   HoldingRegisters[1055] := 16#0000;
   HoldingRegisters[1056] := 16#0000;
   HoldingRegisters[1057] := 16#0000;
   HoldingRegisters[1058] := 16#0000;
   HoldingRegisters[1059] := 16#0000;
   HoldingRegisters[1060] := 16#0000;
   HoldingRegisters[1061] := 16#0000;
   HoldingRegisters[1062] := 16#0000;
   HoldingRegisters[1063] := 16#0000;
   HoldingRegisters[1064] := 16#0000;
   HoldingRegisters[1065] := 16#0000;
   HoldingRegisters[1066] := 16#0000;
   HoldingRegisters[1067] := 16#0000;
   HoldingRegisters[1068] := 16#0000;
   HoldingRegisters[1069] := 16#0000;
   HoldingRegisters[1070] := 16#0000;
   HoldingRegisters[1071] := 16#0000;
   HoldingRegisters[1072] := 16#0000;
   HoldingRegisters[1073] := 16#0000;
   HoldingRegisters[1074] := 16#0000;
   HoldingRegisters[1075] := 16#0000;
   HoldingRegisters[1076] := 16#0000;
   HoldingRegisters[1077] := 16#0000;
   HoldingRegisters[1078] := 16#0000;
   HoldingRegisters[1079] := 16#0000;
   HoldingRegisters[1080] := 16#0000;
   HoldingRegisters[1081] := 16#0000;
   HoldingRegisters[1082] := 16#0000;
   HoldingRegisters[1083] := 16#0000;
   HoldingRegisters[1084] := 16#0000;
   HoldingRegisters[1085] := 16#0000;
   HoldingRegisters[1086] := 16#0000;
   HoldingRegisters[1087] := 16#0000;
   HoldingRegisters[1088] := 16#0000;
   HoldingRegisters[1089] := 16#0000;
   HoldingRegisters[1090] := 16#0000;
   HoldingRegisters[1091] := 16#0000;
   HoldingRegisters[1092] := 16#0000;
   HoldingRegisters[1093] := 16#0000;
   HoldingRegisters[1094] := 16#0000;
   HoldingRegisters[1095] := 16#0000;
   HoldingRegisters[1096] := 16#0000;
   HoldingRegisters[1097] := 16#0000;
   HoldingRegisters[1098] := 16#0000;
   HoldingRegisters[1099] := 16#0000;
   HoldingRegisters[1100] := 16#0000;
   HoldingRegisters[1101] := 16#0000;
   HoldingRegisters[1102] := 16#0000;
   HoldingRegisters[1103] := 16#0000;
   HoldingRegisters[1104] := 16#0000;
   HoldingRegisters[1105] := 16#0000;
   HoldingRegisters[1106] := 16#0000;
   HoldingRegisters[1107] := 16#0000;
   HoldingRegisters[1108] := 16#0000;
   HoldingRegisters[1109] := 16#0000;
   HoldingRegisters[1110] := 16#0000;
   HoldingRegisters[1111] := 16#0000;
   HoldingRegisters[1112] := 16#0000;
   HoldingRegisters[1113] := 16#0000;
   HoldingRegisters[1114] := 16#0000;
   HoldingRegisters[1115] := 16#0000;
   HoldingRegisters[1116] := 16#0000;
   HoldingRegisters[1117] := 16#0000;
   HoldingRegisters[1118] := 16#0000;
   HoldingRegisters[1119] := 16#0000;
   HoldingRegisters[1120] := 16#0000;
   HoldingRegisters[1121] := 16#0000;
   HoldingRegisters[1122] := 16#0000;
   HoldingRegisters[1123] := 16#0000;
   HoldingRegisters[1124] := 16#0000;
   HoldingRegisters[1125] := 16#0000;
   HoldingRegisters[1126] := 16#0000;
   HoldingRegisters[1127] := 16#0000;
   HoldingRegisters[1128] := 16#0000;
   HoldingRegisters[1129] := 16#0000;
   HoldingRegisters[1130] := 16#0000;
   HoldingRegisters[1131] := 16#0000;
   HoldingRegisters[1132] := 16#0000;
   HoldingRegisters[1133] := 16#0000;
   HoldingRegisters[1134] := 16#0000;
   HoldingRegisters[1135] := 16#0000;
   HoldingRegisters[1136] := 16#0000;
   HoldingRegisters[1137] := 16#0000;
   HoldingRegisters[1138] := 16#0000;
   HoldingRegisters[1139] := 16#0000;
   HoldingRegisters[1140] := 16#0000;
   HoldingRegisters[1141] := 16#0000;
   HoldingRegisters[1142] := 16#0000;
   HoldingRegisters[1143] := 16#0000;
   HoldingRegisters[1144] := 16#0000;
   HoldingRegisters[1145] := 16#0000;
   HoldingRegisters[1146] := 16#0000;
   HoldingRegisters[1147] := 16#0000;
   HoldingRegisters[1148] := 16#0000;
   HoldingRegisters[1149] := 16#0000;
   HoldingRegisters[1150] := 16#0000;
   HoldingRegisters[1151] := 16#0000;
   HoldingRegisters[1152] := 16#0000;
   HoldingRegisters[1153] := 16#0000;
   HoldingRegisters[1154] := 16#0000;
   HoldingRegisters[1155] := 16#0000;
   HoldingRegisters[1156] := 16#0000;
   HoldingRegisters[1157] := 16#0000;
   HoldingRegisters[1158] := 16#0000;
   HoldingRegisters[1159] := 16#0000;
   HoldingRegisters[1160] := 16#0000;
   HoldingRegisters[1161] := 16#0000;
   HoldingRegisters[1162] := 16#0000;
   HoldingRegisters[1163] := 16#0000;
   HoldingRegisters[1164] := 16#0000;
   HoldingRegisters[1165] := 16#0000;
   HoldingRegisters[1166] := 16#0000;
   HoldingRegisters[1167] := 16#0000;
   HoldingRegisters[1168] := 16#0000;
   HoldingRegisters[1169] := 16#0000;
   HoldingRegisters[1170] := 16#0000;
   HoldingRegisters[1171] := 16#0000;
   HoldingRegisters[1172] := 16#0000;
   HoldingRegisters[1173] := 16#0000;
   HoldingRegisters[1174] := 16#0000;
   HoldingRegisters[1175] := 16#0000;
   HoldingRegisters[1176] := 16#0000;
   HoldingRegisters[1177] := 16#0000;
   HoldingRegisters[1178] := 16#0000;
   HoldingRegisters[1179] := 16#0000;
   HoldingRegisters[1180] := 16#0000;
   HoldingRegisters[1181] := 16#0000;
   HoldingRegisters[1182] := 16#0000;
   HoldingRegisters[1183] := 16#0000;
   HoldingRegisters[1184] := 16#0000;
   HoldingRegisters[1185] := 16#0000;
   HoldingRegisters[1186] := 16#0000;
   HoldingRegisters[1187] := 16#0000;
   HoldingRegisters[1188] := 16#0000;
   HoldingRegisters[1189] := 16#0000;
   HoldingRegisters[1190] := 16#0000;
   HoldingRegisters[1191] := 16#0000;
   HoldingRegisters[1192] := 16#0000;
   HoldingRegisters[1193] := 16#0000;
   HoldingRegisters[1194] := 16#0000;
   HoldingRegisters[1195] := 16#0000;
   HoldingRegisters[1196] := 16#0000;
   HoldingRegisters[1197] := 16#0000;
   HoldingRegisters[1198] := 16#0000;
   HoldingRegisters[1199] := 16#0000;
   HoldingRegisters[1200] := 16#0000;
   HoldingRegisters[1201] := 16#0000;
   HoldingRegisters[1202] := 16#0000;
   HoldingRegisters[1203] := 16#0000;
   HoldingRegisters[1204] := 16#0000;
   HoldingRegisters[1205] := 16#0000;
   HoldingRegisters[1206] := 16#0000;
   HoldingRegisters[1207] := 16#0000;
   HoldingRegisters[1208] := 16#0000;
   HoldingRegisters[1209] := 16#0000;
   HoldingRegisters[1210] := 16#0000;
   HoldingRegisters[1211] := 16#0000;
   HoldingRegisters[1212] := 16#0000;
   HoldingRegisters[1213] := 16#0000;
   HoldingRegisters[1214] := 16#0000;
   HoldingRegisters[1215] := 16#0000;
   HoldingRegisters[1216] := 16#0000;
   HoldingRegisters[1217] := 16#0000;
   HoldingRegisters[1218] := 16#0000;
   HoldingRegisters[1219] := 16#0000;
   HoldingRegisters[1220] := 16#0000;
   HoldingRegisters[1221] := 16#0000;
   HoldingRegisters[1222] := 16#0000;
   HoldingRegisters[1223] := 16#0000;
   HoldingRegisters[1224] := 16#0000;
   HoldingRegisters[1225] := 16#0000;
   HoldingRegisters[1226] := 16#0000;
   HoldingRegisters[1227] := 16#0000;
   HoldingRegisters[1228] := 16#0000;
   HoldingRegisters[1229] := 16#0000;
   HoldingRegisters[1230] := 16#0000;
   HoldingRegisters[1231] := 16#0000;
   HoldingRegisters[1232] := 16#0000;
   HoldingRegisters[1233] := 16#0000;
   HoldingRegisters[1234] := 16#0000;
   HoldingRegisters[1235] := 16#0000;
   HoldingRegisters[1236] := 16#0000;
   HoldingRegisters[1237] := 16#0000;
   HoldingRegisters[1238] := 16#0000;
   HoldingRegisters[1239] := 16#0000;
   HoldingRegisters[1240] := 16#0000;
   HoldingRegisters[1241] := 16#0000;
   HoldingRegisters[1242] := 16#0000;
   HoldingRegisters[1243] := 16#0000;
   HoldingRegisters[1244] := 16#0000;
   HoldingRegisters[1245] := 16#0000;
   HoldingRegisters[1246] := 16#0000;
   HoldingRegisters[1247] := 16#0000;
   HoldingRegisters[1248] := 16#0000;
   HoldingRegisters[1249] := 16#0000;
   HoldingRegisters[1250] := 16#0000;
   HoldingRegisters[1251] := 16#0000;
   HoldingRegisters[1252] := 16#0000;
   HoldingRegisters[1253] := 16#0000;
   HoldingRegisters[1254] := 16#0000;
   HoldingRegisters[1255] := 16#0000;
   HoldingRegisters[1256] := 16#0000;
   HoldingRegisters[1257] := 16#0000;
   HoldingRegisters[1258] := 16#0000;
   HoldingRegisters[1259] := 16#0000;
   HoldingRegisters[1260] := 16#0000;
   HoldingRegisters[1261] := 16#0000;
   HoldingRegisters[1262] := 16#0000;
   HoldingRegisters[1263] := 16#0000;
   HoldingRegisters[1264] := 16#0000;
   HoldingRegisters[1265] := 16#0000;
   HoldingRegisters[1266] := 16#0000;
   HoldingRegisters[1267] := 16#0000;
   HoldingRegisters[1268] := 16#0000;
   HoldingRegisters[1269] := 16#0000;
   HoldingRegisters[1270] := 16#0000;
   HoldingRegisters[1271] := 16#0000;
   HoldingRegisters[1272] := 16#0000;
   HoldingRegisters[1273] := 16#0000;
   HoldingRegisters[1274] := 16#0000;
   HoldingRegisters[1275] := 16#0000;
   HoldingRegisters[1276] := 16#0000;
   HoldingRegisters[1277] := 16#0000;
   HoldingRegisters[1278] := 16#0000;
   HoldingRegisters[1279] := 16#0000;
   HoldingRegisters[1280] := 16#0000;
   HoldingRegisters[1281] := 16#0000;
   HoldingRegisters[1282] := 16#0000;
   HoldingRegisters[1283] := 16#0000;
   HoldingRegisters[1284] := 16#0000;
   HoldingRegisters[1285] := 16#0000;
   HoldingRegisters[1286] := 16#0000;
   HoldingRegisters[1287] := 16#0000;
   HoldingRegisters[1288] := 16#0000;
   HoldingRegisters[1289] := 16#0000;
   HoldingRegisters[1290] := 16#0000;
   HoldingRegisters[1291] := 16#0000;
   HoldingRegisters[1292] := 16#0000;
   HoldingRegisters[1293] := 16#0000;
   HoldingRegisters[1294] := 16#0000;
   HoldingRegisters[1295] := 16#0000;
   HoldingRegisters[1296] := 16#0000;
   HoldingRegisters[1297] := 16#0000;
   HoldingRegisters[1298] := 16#0000;
   HoldingRegisters[1299] := 16#0000;
   HoldingRegisters[1300] := 16#0000;
   HoldingRegisters[1301] := 16#0000;
   HoldingRegisters[1302] := 16#0000;
   HoldingRegisters[1303] := 16#0000;
   HoldingRegisters[1304] := 16#0000;
   HoldingRegisters[1305] := 16#0000;
   HoldingRegisters[1306] := 16#0000;
   HoldingRegisters[1307] := 16#0000;
   HoldingRegisters[1308] := 16#0000;
   HoldingRegisters[1309] := 16#0000;
   HoldingRegisters[1310] := 16#0000;
   HoldingRegisters[1311] := 16#0000;
   HoldingRegisters[1312] := 16#0000;
   HoldingRegisters[1313] := 16#0000;
   HoldingRegisters[1314] := 16#0000;
   HoldingRegisters[1315] := 16#0000;
   HoldingRegisters[1316] := 16#0000;
   HoldingRegisters[1317] := 16#0000;
   HoldingRegisters[1318] := 16#0000;
   HoldingRegisters[1319] := 16#0000;
   HoldingRegisters[1320] := 16#0000;
   HoldingRegisters[1321] := 16#0000;
   HoldingRegisters[1322] := 16#0000;
   HoldingRegisters[1323] := 16#0000;
   HoldingRegisters[1324] := 16#0000;
   HoldingRegisters[1325] := 16#0000;
   HoldingRegisters[1326] := 16#0000;
   HoldingRegisters[1327] := 16#0000;
   HoldingRegisters[1328] := 16#0000;
   HoldingRegisters[1329] := 16#0000;
   HoldingRegisters[1330] := 16#0000;
   HoldingRegisters[1331] := 16#0000;
   HoldingRegisters[1332] := 16#0000;
   HoldingRegisters[1333] := 16#0000;
   HoldingRegisters[1334] := 16#0000;
   HoldingRegisters[1335] := 16#0000;
   HoldingRegisters[1336] := 16#0000;
   HoldingRegisters[1337] := 16#0000;
   HoldingRegisters[1338] := 16#0000;
   HoldingRegisters[1339] := 16#0000;
   HoldingRegisters[1340] := 16#0000;
   HoldingRegisters[1341] := 16#0000;
   HoldingRegisters[1342] := 16#0000;
   HoldingRegisters[1343] := 16#0000;
   HoldingRegisters[1344] := 16#0000;
   HoldingRegisters[1345] := 16#0000;
   HoldingRegisters[1346] := 16#0000;
   HoldingRegisters[1347] := 16#0000;
   HoldingRegisters[1348] := 16#0000;
   HoldingRegisters[1349] := 16#0000;
   HoldingRegisters[1350] := 16#0000;
   HoldingRegisters[1351] := 16#0000;
   HoldingRegisters[1352] := 16#0000;
   HoldingRegisters[1353] := 16#0000;
   HoldingRegisters[1354] := 16#0000;
   HoldingRegisters[1355] := 16#0000;
   HoldingRegisters[1356] := 16#0000;
   HoldingRegisters[1357] := 16#0000;
   HoldingRegisters[1358] := 16#0000;
   HoldingRegisters[1359] := 16#0000;
   HoldingRegisters[1360] := 16#0000;
   HoldingRegisters[1361] := 16#0000;
   HoldingRegisters[1362] := 16#0000;
   HoldingRegisters[1363] := 16#0000;
   HoldingRegisters[1364] := 16#0000;
   HoldingRegisters[1365] := 16#0000;
   HoldingRegisters[1366] := 16#0000;
   HoldingRegisters[1367] := 16#0000;
   HoldingRegisters[1368] := 16#0000;
   HoldingRegisters[1369] := 16#0000;
   HoldingRegisters[1370] := 16#0000;
   HoldingRegisters[1371] := 16#0000;
   HoldingRegisters[1372] := 16#0000;
   HoldingRegisters[1373] := 16#0000;
   HoldingRegisters[1374] := 16#0000;
   HoldingRegisters[1375] := 16#0000;
   HoldingRegisters[1376] := 16#0000;
   HoldingRegisters[1377] := 16#0000;
   HoldingRegisters[1378] := 16#0000;
   HoldingRegisters[1379] := 16#0000;
   HoldingRegisters[1380] := 16#0000;
   HoldingRegisters[1381] := 16#0000;
   HoldingRegisters[1382] := 16#0000;
   HoldingRegisters[1383] := 16#0000;
   HoldingRegisters[1384] := 16#0000;
   HoldingRegisters[1385] := 16#0000;
   HoldingRegisters[1386] := 16#0000;
   HoldingRegisters[1387] := 16#0000;
   HoldingRegisters[1388] := 16#0000;
   HoldingRegisters[1389] := 16#0000;
   HoldingRegisters[1390] := 16#0000;
   HoldingRegisters[1391] := 16#0000;
   HoldingRegisters[1392] := 16#0000;
   HoldingRegisters[1393] := 16#0000;
   HoldingRegisters[1394] := 16#0000;
   HoldingRegisters[1395] := 16#0000;
   HoldingRegisters[1396] := 16#0000;
   HoldingRegisters[1397] := 16#0000;
   HoldingRegisters[1398] := 16#0000;
   HoldingRegisters[1399] := 16#0000;
   HoldingRegisters[1400] := 16#0000;
   HoldingRegisters[1401] := 16#0000;
   HoldingRegisters[1402] := 16#0000;
   HoldingRegisters[1403] := 16#0000;
   HoldingRegisters[1404] := 16#0000;
   HoldingRegisters[1405] := 16#0000;
   HoldingRegisters[1406] := 16#0000;
   HoldingRegisters[1407] := 16#0000;
   HoldingRegisters[1408] := 16#0000;
   HoldingRegisters[1409] := 16#0000;
   HoldingRegisters[1410] := 16#0000;
   HoldingRegisters[1411] := 16#0000;
   HoldingRegisters[1412] := 16#0000;
   HoldingRegisters[1413] := 16#0000;
   HoldingRegisters[1414] := 16#0000;
   HoldingRegisters[1415] := 16#0000;
   HoldingRegisters[1416] := 16#0000;
   HoldingRegisters[1417] := 16#0000;
   HoldingRegisters[1418] := 16#0000;
   HoldingRegisters[1419] := 16#0000;
   HoldingRegisters[1420] := 16#0000;
   HoldingRegisters[1421] := 16#0000;
   HoldingRegisters[1422] := 16#0000;
   HoldingRegisters[1423] := 16#0000;
   HoldingRegisters[1424] := 16#0000;
   HoldingRegisters[1425] := 16#0000;
   HoldingRegisters[1426] := 16#0000;
   HoldingRegisters[1427] := 16#0000;
   HoldingRegisters[1428] := 16#0000;
   HoldingRegisters[1429] := 16#0000;
   HoldingRegisters[1430] := 16#0000;
   HoldingRegisters[1431] := 16#0000;
   HoldingRegisters[1432] := 16#0000;
   HoldingRegisters[1433] := 16#0000;
   HoldingRegisters[1434] := 16#0000;
   HoldingRegisters[1435] := 16#0000;
   HoldingRegisters[1436] := 16#0000;
   HoldingRegisters[1437] := 16#0000;
   HoldingRegisters[1438] := 16#0000;
   HoldingRegisters[1439] := 16#0000;
   HoldingRegisters[1440] := 16#0000;
   HoldingRegisters[1441] := 16#0000;
   HoldingRegisters[1442] := 16#0000;
   HoldingRegisters[1443] := 16#0000;
   HoldingRegisters[1444] := 16#0000;
   HoldingRegisters[1445] := 16#0000;
   HoldingRegisters[1446] := 16#0000;
   HoldingRegisters[1447] := 16#0000;
   HoldingRegisters[1448] := 16#0000;
   HoldingRegisters[1449] := 16#0000;
   HoldingRegisters[1450] := 16#0000;
   HoldingRegisters[1451] := 16#0000;
   HoldingRegisters[1452] := 16#0000;
   HoldingRegisters[1453] := 16#0000;
   HoldingRegisters[1454] := 16#0000;
   HoldingRegisters[1455] := 16#0000;
   HoldingRegisters[1456] := 16#0000;
   HoldingRegisters[1457] := 16#0000;
   HoldingRegisters[1458] := 16#0000;
   HoldingRegisters[1459] := 16#0000;
   HoldingRegisters[1460] := 16#0000;
   HoldingRegisters[1461] := 16#0000;
   HoldingRegisters[1462] := 16#0000;
   HoldingRegisters[1463] := 16#0000;
   HoldingRegisters[1464] := 16#0000;
   HoldingRegisters[1465] := 16#0000;
   HoldingRegisters[1466] := 16#0000;
   HoldingRegisters[1467] := 16#0000;
   HoldingRegisters[1468] := 16#0000;
   HoldingRegisters[1469] := 16#0000;
   HoldingRegisters[1470] := 16#0000;
   HoldingRegisters[1471] := 16#0000;
   HoldingRegisters[1472] := 16#0000;
   HoldingRegisters[1473] := 16#0000;
   HoldingRegisters[1474] := 16#0000;
   HoldingRegisters[1475] := 16#0000;
   HoldingRegisters[1476] := 16#0000;
   HoldingRegisters[1477] := 16#0000;
   HoldingRegisters[1478] := 16#0000;
   HoldingRegisters[1479] := 16#0000;
   HoldingRegisters[1480] := 16#0000;
   HoldingRegisters[1481] := 16#0000;
   HoldingRegisters[1482] := 16#0000;
   HoldingRegisters[1483] := 16#0000;
   HoldingRegisters[1484] := 16#0000;
   HoldingRegisters[1485] := 16#0000;
   HoldingRegisters[1486] := 16#0000;
   HoldingRegisters[1487] := 16#0000;
   HoldingRegisters[1488] := 16#0000;
   HoldingRegisters[1489] := 16#0000;
   HoldingRegisters[1490] := 16#0000;
   HoldingRegisters[1491] := 16#0000;
   HoldingRegisters[1492] := 16#0000;
   HoldingRegisters[1493] := 16#0000;
   HoldingRegisters[1494] := 16#0000;
   HoldingRegisters[1495] := 16#0000;
   HoldingRegisters[1496] := 16#0000;
   HoldingRegisters[1497] := 16#0000;
   HoldingRegisters[1498] := 16#0000;
   HoldingRegisters[1499] := 16#0000;
   HoldingRegisters[1500] := 16#0000;
   HoldingRegisters[1501] := 16#0000;
   HoldingRegisters[1502] := 16#0000;
   HoldingRegisters[1503] := 16#0000;
   HoldingRegisters[1504] := 16#0000;
   HoldingRegisters[1505] := 16#0000;
   HoldingRegisters[1506] := 16#0000;
   HoldingRegisters[1507] := 16#0000;
   HoldingRegisters[1508] := 16#0000;
   HoldingRegisters[1509] := 16#0000;
   HoldingRegisters[1510] := 16#0000;
   HoldingRegisters[1511] := 16#0000;
   HoldingRegisters[1512] := 16#0000;
   HoldingRegisters[1513] := 16#0000;
   HoldingRegisters[1514] := 16#0000;
   HoldingRegisters[1515] := 16#0000;
   HoldingRegisters[1516] := 16#0000;
   HoldingRegisters[1517] := 16#0000;
   HoldingRegisters[1518] := 16#0000;
   HoldingRegisters[1519] := 16#0000;
   HoldingRegisters[1520] := 16#0000;
   HoldingRegisters[1521] := 16#0000;
   HoldingRegisters[1522] := 16#0000;
   HoldingRegisters[1523] := 16#0000;
   HoldingRegisters[1524] := 16#0000;
   HoldingRegisters[1525] := 16#0000;
   HoldingRegisters[1526] := 16#0000;
   HoldingRegisters[1527] := 16#0000;
   HoldingRegisters[1528] := 16#0000;
   HoldingRegisters[1529] := 16#0000;
   HoldingRegisters[1530] := 16#0000;
   HoldingRegisters[1531] := 16#0000;
   HoldingRegisters[1532] := 16#0000;
   HoldingRegisters[1533] := 16#0000;
   HoldingRegisters[1534] := 16#0000;
   HoldingRegisters[1535] := 16#0000;
   HoldingRegisters[1536] := 16#0000;
   HoldingRegisters[1537] := 16#0000;
   HoldingRegisters[1538] := 16#0000;
   HoldingRegisters[1539] := 16#0000;
   HoldingRegisters[1540] := 16#0000;
   HoldingRegisters[1541] := 16#0000;
   HoldingRegisters[1542] := 16#0000;
   HoldingRegisters[1543] := 16#0000;
   HoldingRegisters[1544] := 16#0000;
   HoldingRegisters[1545] := 16#0000;
   HoldingRegisters[1546] := 16#0000;
   HoldingRegisters[1547] := 16#0000;
   HoldingRegisters[1548] := 16#0000;
   HoldingRegisters[1549] := 16#0000;
   HoldingRegisters[1550] := 16#0000;
   HoldingRegisters[1551] := 16#0000;
   HoldingRegisters[1552] := 16#0000;
   HoldingRegisters[1553] := 16#0000;
   HoldingRegisters[1554] := 16#0000;
   HoldingRegisters[1555] := 16#0000;
   HoldingRegisters[1556] := 16#0000;
   HoldingRegisters[1557] := 16#0000;
   HoldingRegisters[1558] := 16#0000;
   HoldingRegisters[1559] := 16#0000;
   HoldingRegisters[1560] := 16#0000;
   HoldingRegisters[1561] := 16#0000;
   HoldingRegisters[1562] := 16#0000;
   HoldingRegisters[1563] := 16#0000;
   HoldingRegisters[1564] := 16#0000;
   HoldingRegisters[1565] := 16#0000;
   HoldingRegisters[1566] := 16#0000;
   HoldingRegisters[1567] := 16#0000;
   HoldingRegisters[1568] := 16#0000;
   HoldingRegisters[1569] := 16#0000;
   HoldingRegisters[1570] := 16#0000;
   HoldingRegisters[1571] := 16#0000;
   HoldingRegisters[1572] := 16#0000;
   HoldingRegisters[1573] := 16#0000;
   HoldingRegisters[1574] := 16#0000;
   HoldingRegisters[1575] := 16#0000;
   HoldingRegisters[1576] := 16#0000;
   HoldingRegisters[1577] := 16#0000;
   HoldingRegisters[1578] := 16#0000;
   HoldingRegisters[1579] := 16#0000;
   HoldingRegisters[1580] := 16#0000;
   HoldingRegisters[1581] := 16#0000;
   HoldingRegisters[1582] := 16#0000;
   HoldingRegisters[1583] := 16#0000;
   HoldingRegisters[1584] := 16#0000;
   HoldingRegisters[1585] := 16#0000;
   HoldingRegisters[1586] := 16#0000;
   HoldingRegisters[1587] := 16#0000;
   HoldingRegisters[1588] := 16#0000;
   HoldingRegisters[1589] := 16#0000;
   HoldingRegisters[1590] := 16#0000;
   HoldingRegisters[1591] := 16#0000;
   HoldingRegisters[1592] := 16#0000;
   HoldingRegisters[1593] := 16#0000;
   HoldingRegisters[1594] := 16#0000;
   HoldingRegisters[1595] := 16#0000;
   HoldingRegisters[1596] := 16#0000;
   HoldingRegisters[1597] := 16#0000;
   HoldingRegisters[1598] := 16#0000;
   HoldingRegisters[1599] := 16#0000;
   HoldingRegisters[1600] := 16#0000;
   HoldingRegisters[1601] := 16#0000;
   HoldingRegisters[1602] := 16#0000;
   HoldingRegisters[1603] := 16#0000;
   HoldingRegisters[1604] := 16#0000;
   HoldingRegisters[1605] := 16#0000;
   HoldingRegisters[1606] := 16#0000;
   HoldingRegisters[1607] := 16#0000;
   HoldingRegisters[1608] := 16#0000;
   HoldingRegisters[1609] := 16#0000;
   HoldingRegisters[1610] := 16#0000;
   HoldingRegisters[1611] := 16#0000;
   HoldingRegisters[1612] := 16#0000;
   HoldingRegisters[1613] := 16#0000;
   HoldingRegisters[1614] := 16#0000;
   HoldingRegisters[1615] := 16#0000;
   HoldingRegisters[1616] := 16#0000;
   HoldingRegisters[1617] := 16#0000;
   HoldingRegisters[1618] := 16#0000;
   HoldingRegisters[1619] := 16#0000;
   HoldingRegisters[1620] := 16#0000;
   HoldingRegisters[1621] := 16#0000;
   HoldingRegisters[1622] := 16#0000;
   HoldingRegisters[1623] := 16#0000;
   HoldingRegisters[1624] := 16#0000;
   HoldingRegisters[1625] := 16#0000;
   HoldingRegisters[1626] := 16#0000;
   HoldingRegisters[1627] := 16#0000;
   HoldingRegisters[1628] := 16#0000;
   HoldingRegisters[1629] := 16#0000;
   HoldingRegisters[1630] := 16#0000;
   HoldingRegisters[1631] := 16#0000;
   HoldingRegisters[1632] := 16#0000;
   HoldingRegisters[1633] := 16#0000;
   HoldingRegisters[1634] := 16#0000;
   HoldingRegisters[1635] := 16#0000;
   HoldingRegisters[1636] := 16#0000;
   HoldingRegisters[1637] := 16#0000;
   HoldingRegisters[1638] := 16#0000;
   HoldingRegisters[1639] := 16#0000;
   HoldingRegisters[1640] := 16#0000;
   HoldingRegisters[1641] := 16#0000;
   HoldingRegisters[1642] := 16#0000;
   HoldingRegisters[1643] := 16#0000;
   HoldingRegisters[1644] := 16#0000;
   HoldingRegisters[1645] := 16#0000;
   HoldingRegisters[1646] := 16#0000;
   HoldingRegisters[1647] := 16#0000;
   HoldingRegisters[1648] := 16#0000;
   HoldingRegisters[1649] := 16#0000;
   HoldingRegisters[1650] := 16#0000;
   HoldingRegisters[1651] := 16#0000;
   HoldingRegisters[1652] := 16#0000;
   HoldingRegisters[1653] := 16#0000;
   HoldingRegisters[1654] := 16#0000;
   HoldingRegisters[1655] := 16#0000;
   HoldingRegisters[1656] := 16#0000;
   HoldingRegisters[1657] := 16#0000;
   HoldingRegisters[1658] := 16#0000;
   HoldingRegisters[1659] := 16#0000;
   HoldingRegisters[1660] := 16#0000;
   HoldingRegisters[1661] := 16#0000;
   HoldingRegisters[1662] := 16#0000;
   HoldingRegisters[1663] := 16#0000;
   HoldingRegisters[1664] := 16#0000;
   HoldingRegisters[1665] := 16#0000;
   HoldingRegisters[1666] := 16#0000;
   HoldingRegisters[1667] := 16#0000;
   HoldingRegisters[1668] := 16#0000;
   HoldingRegisters[1669] := 16#0000;
   HoldingRegisters[1670] := 16#0000;
   HoldingRegisters[1671] := 16#0000;
   HoldingRegisters[1672] := 16#0000;
   HoldingRegisters[1673] := 16#0000;
   HoldingRegisters[1674] := 16#0000;
   HoldingRegisters[1675] := 16#0000;
   HoldingRegisters[1676] := 16#0000;
   HoldingRegisters[1677] := 16#0000;
   HoldingRegisters[1678] := 16#0000;
   HoldingRegisters[1679] := 16#0000;
   HoldingRegisters[1680] := 16#0000;
   HoldingRegisters[1681] := 16#0000;
   HoldingRegisters[1682] := 16#0000;
   HoldingRegisters[1683] := 16#0000;
   HoldingRegisters[1684] := 16#0000;
   HoldingRegisters[1685] := 16#0000;
   HoldingRegisters[1686] := 16#0000;
   HoldingRegisters[1687] := 16#0000;
   HoldingRegisters[1688] := 16#0000;
   HoldingRegisters[1689] := 16#0000;
   HoldingRegisters[1690] := 16#0000;
   HoldingRegisters[1691] := 16#0000;
   HoldingRegisters[1692] := 16#0000;
   HoldingRegisters[1693] := 16#0000;
   HoldingRegisters[1694] := 16#0000;
   HoldingRegisters[1695] := 16#0000;
   HoldingRegisters[1696] := 16#0000;
   HoldingRegisters[1697] := 16#0000;
   HoldingRegisters[1698] := 16#0000;
   HoldingRegisters[1699] := 16#0000;
   HoldingRegisters[1700] := 16#0000;
   HoldingRegisters[1701] := 16#0000;
   HoldingRegisters[1702] := 16#0000;
   HoldingRegisters[1703] := 16#0000;
   HoldingRegisters[1704] := 16#0000;
   HoldingRegisters[1705] := 16#0000;
   HoldingRegisters[1706] := 16#0000;
   HoldingRegisters[1707] := 16#0000;
   HoldingRegisters[1708] := 16#0000;
   HoldingRegisters[1709] := 16#0000;
   HoldingRegisters[1710] := 16#0000;
   HoldingRegisters[1711] := 16#0000;
   HoldingRegisters[1712] := 16#0000;
   HoldingRegisters[1713] := 16#0000;
   HoldingRegisters[1714] := 16#0000;
   HoldingRegisters[1715] := 16#0000;
   HoldingRegisters[1716] := 16#0000;
   HoldingRegisters[1717] := 16#0000;
   HoldingRegisters[1718] := 16#0000;
   HoldingRegisters[1719] := 16#0000;
   HoldingRegisters[1720] := 16#0000;
   HoldingRegisters[1721] := 16#0000;
   HoldingRegisters[1722] := 16#0000;
   HoldingRegisters[1723] := 16#0000;
   HoldingRegisters[1724] := 16#0000;
   HoldingRegisters[1725] := 16#0000;
   HoldingRegisters[1726] := 16#0000;
   HoldingRegisters[1727] := 16#0000;
   HoldingRegisters[1728] := 16#0000;
   HoldingRegisters[1729] := 16#0000;
   HoldingRegisters[1730] := 16#0000;
   HoldingRegisters[1731] := 16#0000;
   HoldingRegisters[1732] := 16#0000;
   HoldingRegisters[1733] := 16#0000;
   HoldingRegisters[1734] := 16#0000;
   HoldingRegisters[1735] := 16#0000;
   HoldingRegisters[1736] := 16#0000;
   HoldingRegisters[1737] := 16#0000;
   HoldingRegisters[1738] := 16#0000;
   HoldingRegisters[1739] := 16#0000;
   HoldingRegisters[1740] := 16#0000;
   HoldingRegisters[1741] := 16#0000;
   HoldingRegisters[1742] := 16#0000;
   HoldingRegisters[1743] := 16#0000;
   HoldingRegisters[1744] := 16#0000;
   HoldingRegisters[1745] := 16#0000;
   HoldingRegisters[1746] := 16#0000;
   HoldingRegisters[1747] := 16#0000;
   HoldingRegisters[1748] := 16#0000;
   HoldingRegisters[1749] := 16#0000;
   HoldingRegisters[1750] := 16#0000;
   HoldingRegisters[1751] := 16#0000;
   HoldingRegisters[1752] := 16#0000;
   HoldingRegisters[1753] := 16#0000;
   HoldingRegisters[1754] := 16#0000;
   HoldingRegisters[1755] := 16#0000;
   HoldingRegisters[1756] := 16#0000;
   HoldingRegisters[1757] := 16#0000;
   HoldingRegisters[1758] := 16#0000;
   HoldingRegisters[1759] := 16#0000;
   HoldingRegisters[1760] := 16#0000;
   HoldingRegisters[1761] := 16#0000;
   HoldingRegisters[1762] := 16#0000;
   HoldingRegisters[1763] := 16#0000;
   HoldingRegisters[1764] := 16#0000;
   HoldingRegisters[1765] := 16#0000;
   HoldingRegisters[1766] := 16#0000;
   HoldingRegisters[1767] := 16#0000;
   HoldingRegisters[1768] := 16#0000;
   HoldingRegisters[1769] := 16#0000;
   HoldingRegisters[1770] := 16#0000;
   HoldingRegisters[1771] := 16#0000;
   HoldingRegisters[1772] := 16#0000;
   HoldingRegisters[1773] := 16#0000;
   HoldingRegisters[1774] := 16#0000;
   HoldingRegisters[1775] := 16#0000;
   HoldingRegisters[1776] := 16#0000;
   HoldingRegisters[1777] := 16#0000;
   HoldingRegisters[1778] := 16#0000;
   HoldingRegisters[1779] := 16#0000;
   HoldingRegisters[1780] := 16#0000;
   HoldingRegisters[1781] := 16#0000;
   HoldingRegisters[1782] := 16#0000;
   HoldingRegisters[1783] := 16#0000;
   HoldingRegisters[1784] := 16#0000;
   HoldingRegisters[1785] := 16#0000;
   HoldingRegisters[1786] := 16#0000;
   HoldingRegisters[1787] := 16#0000;
   HoldingRegisters[1788] := 16#0000;
   HoldingRegisters[1789] := 16#0000;
   HoldingRegisters[1790] := 16#0000;
   HoldingRegisters[1791] := 16#0000;
   HoldingRegisters[1792] := 16#0000;
   HoldingRegisters[1793] := 16#0000;
   HoldingRegisters[1794] := 16#0000;
   HoldingRegisters[1795] := 16#0000;
   HoldingRegisters[1796] := 16#0000;
   HoldingRegisters[1797] := 16#0000;
   HoldingRegisters[1798] := 16#0000;
   HoldingRegisters[1799] := 16#0000;
   HoldingRegisters[1800] := 16#0000;
   HoldingRegisters[1801] := 16#0000;
   HoldingRegisters[1802] := 16#0000;
   HoldingRegisters[1803] := 16#0000;
   HoldingRegisters[1804] := 16#0000;
   HoldingRegisters[1805] := 16#0000;
   HoldingRegisters[1806] := 16#0000;
   HoldingRegisters[1807] := 16#0000;
   HoldingRegisters[1808] := 16#0000;
   HoldingRegisters[1809] := 16#0000;
   HoldingRegisters[1810] := 16#0000;
   HoldingRegisters[1811] := 16#0000;
   HoldingRegisters[1812] := 16#0000;
   HoldingRegisters[1813] := 16#0000;
   HoldingRegisters[1814] := 16#0000;
   HoldingRegisters[1815] := 16#0000;
   HoldingRegisters[1816] := 16#0000;
   HoldingRegisters[1817] := 16#0000;
   HoldingRegisters[1818] := 16#0000;
   HoldingRegisters[1819] := 16#0000;
   HoldingRegisters[1820] := 16#0000;
   HoldingRegisters[1821] := 16#0000;
   HoldingRegisters[1822] := 16#0000;
   HoldingRegisters[1823] := 16#0000;
   HoldingRegisters[1824] := 16#0000;
   HoldingRegisters[1825] := 16#0000;
   HoldingRegisters[1826] := 16#0000;
   HoldingRegisters[1827] := 16#0000;
   HoldingRegisters[1828] := 16#0000;
   HoldingRegisters[1829] := 16#0000;
   HoldingRegisters[1830] := 16#0000;
   HoldingRegisters[1831] := 16#0000;
   HoldingRegisters[1832] := 16#0000;
   HoldingRegisters[1833] := 16#0000;
   HoldingRegisters[1834] := 16#0000;
   HoldingRegisters[1835] := 16#0000;
   HoldingRegisters[1836] := 16#0000;
   HoldingRegisters[1837] := 16#0000;
   HoldingRegisters[1838] := 16#0000;
   HoldingRegisters[1839] := 16#0000;
   HoldingRegisters[1840] := 16#0000;
   HoldingRegisters[1841] := 16#0000;
   HoldingRegisters[1842] := 16#0000;
   HoldingRegisters[1843] := 16#0000;
   HoldingRegisters[1844] := 16#0000;
   HoldingRegisters[1845] := 16#0000;
   HoldingRegisters[1846] := 16#0000;
   HoldingRegisters[1847] := 16#0000;
   HoldingRegisters[1848] := 16#0000;
   HoldingRegisters[1849] := 16#0000;
   HoldingRegisters[1850] := 16#0000;
   HoldingRegisters[1851] := 16#0000;
   HoldingRegisters[1852] := 16#0000;
   HoldingRegisters[1853] := 16#0000;
   HoldingRegisters[1854] := 16#0000;
   HoldingRegisters[1855] := 16#0000;
   HoldingRegisters[1856] := 16#0000;
   HoldingRegisters[1857] := 16#0000;
   HoldingRegisters[1858] := 16#0000;
   HoldingRegisters[1859] := 16#0000;
   HoldingRegisters[1860] := 16#0000;
   HoldingRegisters[1861] := 16#0000;
   HoldingRegisters[1862] := 16#0000;
   HoldingRegisters[1863] := 16#0000;
   HoldingRegisters[1864] := 16#0000;
   HoldingRegisters[1865] := 16#0000;
   HoldingRegisters[1866] := 16#0000;
   HoldingRegisters[1867] := 16#0000;
   HoldingRegisters[1868] := 16#0000;
   HoldingRegisters[1869] := 16#0000;
   HoldingRegisters[1870] := 16#0000;
   HoldingRegisters[1871] := 16#0000;
   HoldingRegisters[1872] := 16#0000;
   HoldingRegisters[1873] := 16#0000;
   HoldingRegisters[1874] := 16#0000;
   HoldingRegisters[1875] := 16#0000;
   HoldingRegisters[1876] := 16#0000;
   HoldingRegisters[1877] := 16#0000;
   HoldingRegisters[1878] := 16#0000;
   HoldingRegisters[1879] := 16#0000;
   HoldingRegisters[1880] := 16#0000;
   HoldingRegisters[1881] := 16#0000;
   HoldingRegisters[1882] := 16#0000;
   HoldingRegisters[1883] := 16#0000;
   HoldingRegisters[1884] := 16#0000;
   HoldingRegisters[1885] := 16#0000;
   HoldingRegisters[1886] := 16#0000;
   HoldingRegisters[1887] := 16#0000;
   HoldingRegisters[1888] := 16#0000;
   HoldingRegisters[1889] := 16#0000;
   HoldingRegisters[1890] := 16#0000;
   HoldingRegisters[1891] := 16#0000;
   HoldingRegisters[1892] := 16#0000;
   HoldingRegisters[1893] := 16#0000;
   HoldingRegisters[1894] := 16#0000;
   HoldingRegisters[1895] := 16#0000;
   HoldingRegisters[1896] := 16#0000;
   HoldingRegisters[1897] := 16#0000;
   HoldingRegisters[1898] := 16#0000;
   HoldingRegisters[1899] := 16#0000;
   HoldingRegisters[1900] := 16#0000;
   HoldingRegisters[1901] := 16#0000;
   HoldingRegisters[1902] := 16#0000;
   HoldingRegisters[1903] := 16#0000;
   HoldingRegisters[1904] := 16#0000;
   HoldingRegisters[1905] := 16#0000;
   HoldingRegisters[1906] := 16#0000;
   HoldingRegisters[1907] := 16#0000;
   HoldingRegisters[1908] := 16#0000;
   HoldingRegisters[1909] := 16#0000;
   HoldingRegisters[1910] := 16#0000;
   HoldingRegisters[1911] := 16#0000;
   HoldingRegisters[1912] := 16#0000;
   HoldingRegisters[1913] := 16#0000;
   HoldingRegisters[1914] := 16#0000;
   HoldingRegisters[1915] := 16#0000;
   HoldingRegisters[1916] := 16#0000;
   HoldingRegisters[1917] := 16#0000;
   HoldingRegisters[1918] := 16#0000;
   HoldingRegisters[1919] := 16#0000;
   HoldingRegisters[1920] := 16#0000;
   HoldingRegisters[1921] := 16#0000;
   HoldingRegisters[1922] := 16#0000;
   HoldingRegisters[1923] := 16#0000;
   HoldingRegisters[1924] := 16#0000;
   HoldingRegisters[1925] := 16#0000;
   HoldingRegisters[1926] := 16#0000;
   HoldingRegisters[1927] := 16#0000;
   HoldingRegisters[1928] := 16#0000;
   HoldingRegisters[1929] := 16#0000;
   HoldingRegisters[1930] := 16#0000;
   HoldingRegisters[1931] := 16#0000;
   HoldingRegisters[1932] := 16#0000;
   HoldingRegisters[1933] := 16#0000;
   HoldingRegisters[1934] := 16#0000;
   HoldingRegisters[1935] := 16#0000;
   HoldingRegisters[1936] := 16#0000;
   HoldingRegisters[1937] := 16#0000;
   HoldingRegisters[1938] := 16#0000;
   HoldingRegisters[1939] := 16#0000;
   HoldingRegisters[1940] := 16#0000;
   HoldingRegisters[1941] := 16#0000;
   HoldingRegisters[1942] := 16#0000;
   HoldingRegisters[1943] := 16#0000;
   HoldingRegisters[1944] := 16#0000;
   HoldingRegisters[1945] := 16#0000;
   HoldingRegisters[1946] := 16#0000;
   HoldingRegisters[1947] := 16#0000;
   HoldingRegisters[1948] := 16#0000;
   HoldingRegisters[1949] := 16#0000;
   HoldingRegisters[1950] := 16#0000;
   HoldingRegisters[1951] := 16#0000;
   HoldingRegisters[1952] := 16#0000;
   HoldingRegisters[1953] := 16#0000;
   HoldingRegisters[1954] := 16#0000;
   HoldingRegisters[1955] := 16#0000;
   HoldingRegisters[1956] := 16#0000;
   HoldingRegisters[1957] := 16#0000;
   HoldingRegisters[1958] := 16#0000;
   HoldingRegisters[1959] := 16#0000;
   HoldingRegisters[1960] := 16#0000;
   HoldingRegisters[1961] := 16#0000;
   HoldingRegisters[1962] := 16#0000;
   HoldingRegisters[1963] := 16#0000;
   HoldingRegisters[1964] := 16#0000;
   HoldingRegisters[1965] := 16#0000;
   HoldingRegisters[1966] := 16#0000;
   HoldingRegisters[1967] := 16#0000;
   HoldingRegisters[1968] := 16#0000;
   HoldingRegisters[1969] := 16#0000;
   HoldingRegisters[1970] := 16#0000;
   HoldingRegisters[1971] := 16#0000;
   HoldingRegisters[1972] := 16#0000;
   HoldingRegisters[1973] := 16#0000;
   HoldingRegisters[1974] := 16#0000;
   HoldingRegisters[1975] := 16#0000;
   HoldingRegisters[1976] := 16#0000;
   HoldingRegisters[1977] := 16#0000;
   HoldingRegisters[1978] := 16#0000;
   HoldingRegisters[1979] := 16#0000;
   HoldingRegisters[1980] := 16#0000;
   HoldingRegisters[1981] := 16#0000;
   HoldingRegisters[1982] := 16#0000;
   HoldingRegisters[1983] := 16#0000;
   HoldingRegisters[1984] := 16#0000;
   HoldingRegisters[1985] := 16#0000;
   HoldingRegisters[1986] := 16#0000;
   HoldingRegisters[1987] := 16#0000;
   HoldingRegisters[1988] := 16#0000;
   HoldingRegisters[1989] := 16#0000;
   HoldingRegisters[1990] := 16#0000;
   HoldingRegisters[1991] := 16#0000;
   HoldingRegisters[1992] := 16#0000;
   HoldingRegisters[1993] := 16#0000;
   HoldingRegisters[1994] := 16#0000;
   HoldingRegisters[1995] := 16#0000;
   HoldingRegisters[1996] := 16#0000;
   HoldingRegisters[1997] := 16#0000;
   HoldingRegisters[1998] := 16#0000;
   HoldingRegisters[1999] := 16#0000;
   HoldingRegisters[2000] := 16#0000;
   HoldingRegisters[2001] := 16#0000;
   HoldingRegisters[2002] := 16#0000;
   HoldingRegisters[2003] := 16#0000;
   HoldingRegisters[2004] := 16#0000;
   HoldingRegisters[2005] := 16#0000;
   HoldingRegisters[2006] := 16#0000;
   HoldingRegisters[2007] := 16#0000;
   HoldingRegisters[2008] := 16#0000;
   HoldingRegisters[2009] := 16#0000;
   HoldingRegisters[2010] := 16#0000;
   HoldingRegisters[2011] := 16#0000;
   HoldingRegisters[2012] := 16#0000;
   HoldingRegisters[2013] := 16#0000;
   HoldingRegisters[2014] := 16#0000;
   HoldingRegisters[2015] := 16#0000;
   HoldingRegisters[2016] := 16#0000;
   HoldingRegisters[2017] := 16#0000;
   HoldingRegisters[2018] := 16#0000;
   HoldingRegisters[2019] := 16#0000;
   HoldingRegisters[2020] := 16#0000;
   HoldingRegisters[2021] := 16#0000;
   HoldingRegisters[2022] := 16#0000;
   HoldingRegisters[2023] := 16#0000;
   HoldingRegisters[2024] := 16#0000;
   HoldingRegisters[2025] := 16#0000;
   HoldingRegisters[2026] := 16#0000;
   HoldingRegisters[2027] := 16#0000;
   HoldingRegisters[2028] := 16#0000;
   HoldingRegisters[2029] := 16#0000;
   HoldingRegisters[2030] := 16#0000;
   HoldingRegisters[2031] := 16#0000;
   HoldingRegisters[2032] := 16#0000;
   HoldingRegisters[2033] := 16#0000;
   HoldingRegisters[2034] := 16#0000;
   HoldingRegisters[2035] := 16#0000;
   HoldingRegisters[2036] := 16#0000;
   HoldingRegisters[2037] := 16#0000;
   HoldingRegisters[2038] := 16#0000;
   HoldingRegisters[2039] := 16#0000;
   HoldingRegisters[2040] := 16#0000;
   HoldingRegisters[2041] := 16#0000;
   HoldingRegisters[2042] := 16#0000;
   HoldingRegisters[2043] := 16#0000;
   HoldingRegisters[2044] := 16#0000;
   HoldingRegisters[2045] := 16#0000;
   HoldingRegisters[2046] := 16#0000;
   HoldingRegisters[2047] := 16#0000;
   HoldingRegisters[2048] := 16#0000;
   HoldingRegisters[2049] := 16#0000;
   HoldingRegisters[2050] := 16#0000;
   HoldingRegisters[2051] := 16#0000;
   HoldingRegisters[2052] := 16#0000;
   HoldingRegisters[2053] := 16#0000;
   HoldingRegisters[2054] := 16#0000;
   HoldingRegisters[2055] := 16#0000;
   HoldingRegisters[2056] := 16#0000;
   HoldingRegisters[2057] := 16#0000;
   HoldingRegisters[2058] := 16#0000;
   HoldingRegisters[2059] := 16#0000;
   HoldingRegisters[2060] := 16#0000;
   HoldingRegisters[2061] := 16#0000;
   HoldingRegisters[2062] := 16#0000;
   HoldingRegisters[2063] := 16#0000;
   HoldingRegisters[2064] := 16#0000;
   HoldingRegisters[2065] := 16#0000;
   HoldingRegisters[2066] := 16#0000;
   HoldingRegisters[2067] := 16#0000;
   HoldingRegisters[2068] := 16#0000;
   HoldingRegisters[2069] := 16#0000;
   HoldingRegisters[2070] := 16#0000;
   HoldingRegisters[2071] := 16#0000;
   HoldingRegisters[2072] := 16#0000;
   HoldingRegisters[2073] := 16#0000;
   HoldingRegisters[2074] := 16#0000;
   HoldingRegisters[2075] := 16#0000;
   HoldingRegisters[2076] := 16#0000;
   HoldingRegisters[2077] := 16#0000;
   HoldingRegisters[2078] := 16#0000;
   HoldingRegisters[2079] := 16#0000;
   HoldingRegisters[2080] := 16#0000;
   HoldingRegisters[2081] := 16#0000;
   HoldingRegisters[2082] := 16#0000;
   HoldingRegisters[2083] := 16#0000;
   HoldingRegisters[2084] := 16#0000;
   HoldingRegisters[2085] := 16#0000;
   HoldingRegisters[2086] := 16#0000;
   HoldingRegisters[2087] := 16#0000;
   HoldingRegisters[2088] := 16#0000;
   HoldingRegisters[2089] := 16#0000;
   HoldingRegisters[2090] := 16#0000;
   HoldingRegisters[2091] := 16#0000;
   HoldingRegisters[2092] := 16#0000;
   HoldingRegisters[2093] := 16#0000;
   HoldingRegisters[2094] := 16#0000;
   HoldingRegisters[2095] := 16#0000;
   HoldingRegisters[2096] := 16#0000;
   HoldingRegisters[2097] := 16#0000;
   HoldingRegisters[2098] := 16#0000;
   HoldingRegisters[2099] := 16#0000;
   HoldingRegisters[2100] := 16#0000;
   HoldingRegisters[2101] := 16#0000;
   HoldingRegisters[2102] := 16#0000;
   HoldingRegisters[2103] := 16#0000;
   HoldingRegisters[2104] := 16#0000;
   HoldingRegisters[2105] := 16#0000;
   HoldingRegisters[2106] := 16#0000;
   HoldingRegisters[2107] := 16#0000;
   HoldingRegisters[2108] := 16#0000;
   HoldingRegisters[2109] := 16#0000;
   HoldingRegisters[2110] := 16#0000;
   HoldingRegisters[2111] := 16#0000;
   HoldingRegisters[2112] := 16#0000;
   HoldingRegisters[2113] := 16#0000;
   HoldingRegisters[2114] := 16#0000;
   HoldingRegisters[2115] := 16#0000;
   HoldingRegisters[2116] := 16#0000;
   HoldingRegisters[2117] := 16#0000;
   HoldingRegisters[2118] := 16#0000;
   HoldingRegisters[2119] := 16#0000;
   HoldingRegisters[2120] := 16#0000;
   HoldingRegisters[2121] := 16#0000;
   HoldingRegisters[2122] := 16#0000;
   HoldingRegisters[2123] := 16#0000;
   HoldingRegisters[2124] := 16#0000;
   HoldingRegisters[2125] := 16#0000;
   HoldingRegisters[2126] := 16#0000;
   HoldingRegisters[2127] := 16#0000;
   HoldingRegisters[2128] := 16#0000;
   HoldingRegisters[2129] := 16#0000;
   HoldingRegisters[2130] := 16#0000;
   HoldingRegisters[2131] := 16#0000;
   HoldingRegisters[2132] := 16#0000;
   HoldingRegisters[2133] := 16#0000;
   HoldingRegisters[2134] := 16#0000;
   HoldingRegisters[2135] := 16#0000;
   HoldingRegisters[2136] := 16#0000;
   HoldingRegisters[2137] := 16#0000;
   HoldingRegisters[2138] := 16#0000;
   HoldingRegisters[2139] := 16#0000;
   HoldingRegisters[2140] := 16#0000;
   HoldingRegisters[2141] := 16#0000;
   HoldingRegisters[2142] := 16#0000;
   HoldingRegisters[2143] := 16#0000;
   HoldingRegisters[2144] := 16#0000;
   HoldingRegisters[2145] := 16#0000;
   HoldingRegisters[2146] := 16#0000;
   HoldingRegisters[2147] := 16#0000;
   HoldingRegisters[2148] := 16#0000;
   HoldingRegisters[2149] := 16#0000;
   HoldingRegisters[2150] := 16#0000;
   HoldingRegisters[2151] := 16#0000;
   HoldingRegisters[2152] := 16#0000;
   HoldingRegisters[2153] := 16#0000;
   HoldingRegisters[2154] := 16#0000;
   HoldingRegisters[2155] := 16#0000;
   HoldingRegisters[2156] := 16#0000;
   HoldingRegisters[2157] := 16#0000;
   HoldingRegisters[2158] := 16#0000;
   HoldingRegisters[2159] := 16#0000;
   HoldingRegisters[2160] := 16#0000;
   HoldingRegisters[2161] := 16#0000;
   HoldingRegisters[2162] := 16#0000;
   HoldingRegisters[2163] := 16#0000;
   HoldingRegisters[2164] := 16#0000;
   HoldingRegisters[2165] := 16#0000;
   HoldingRegisters[2166] := 16#0000;
   HoldingRegisters[2167] := 16#0000;
   HoldingRegisters[2168] := 16#0000;
   HoldingRegisters[2169] := 16#0000;
   HoldingRegisters[2170] := 16#0000;
   HoldingRegisters[2171] := 16#0000;
   HoldingRegisters[2172] := 16#0000;
   HoldingRegisters[2173] := 16#0000;
   HoldingRegisters[2174] := 16#0000;
   HoldingRegisters[2175] := 16#0000;
   HoldingRegisters[2176] := 16#0000;
   HoldingRegisters[2177] := 16#0000;
   HoldingRegisters[2178] := 16#0000;
   HoldingRegisters[2179] := 16#0000;
   HoldingRegisters[2180] := 16#0000;
   HoldingRegisters[2181] := 16#0000;
   HoldingRegisters[2182] := 16#0000;
   HoldingRegisters[2183] := 16#0000;
   HoldingRegisters[2184] := 16#0000;
   HoldingRegisters[2185] := 16#0000;
   HoldingRegisters[2186] := 16#0000;
   HoldingRegisters[2187] := 16#0000;
   HoldingRegisters[2188] := 16#0000;
   HoldingRegisters[2189] := 16#0000;
   HoldingRegisters[2190] := 16#0000;
   HoldingRegisters[2191] := 16#0000;
   HoldingRegisters[2192] := 16#0000;
   HoldingRegisters[2193] := 16#0000;
   HoldingRegisters[2194] := 16#0000;
   HoldingRegisters[2195] := 16#0000;
   HoldingRegisters[2196] := 16#0000;
   HoldingRegisters[2197] := 16#0000;
   HoldingRegisters[2198] := 16#0000;
   HoldingRegisters[2199] := 16#0000;
   HoldingRegisters[2200] := 16#0000;
   HoldingRegisters[2201] := 16#0000;
   HoldingRegisters[2202] := 16#0000;
   HoldingRegisters[2203] := 16#0000;
   HoldingRegisters[2204] := 16#0000;
   HoldingRegisters[2205] := 16#0000;
   HoldingRegisters[2206] := 16#0000;
   HoldingRegisters[2207] := 16#0000;
   HoldingRegisters[2208] := 16#0000;
   HoldingRegisters[2209] := 16#0000;
   HoldingRegisters[2210] := 16#0000;
   HoldingRegisters[2211] := 16#0000;
   HoldingRegisters[2212] := 16#0000;
   HoldingRegisters[2213] := 16#0000;
   HoldingRegisters[2214] := 16#0000;
   HoldingRegisters[2215] := 16#0000;
   HoldingRegisters[2216] := 16#0000;
   HoldingRegisters[2217] := 16#0000;
   HoldingRegisters[2218] := 16#0000;
   HoldingRegisters[2219] := 16#0000;
   HoldingRegisters[2220] := 16#0000;
   HoldingRegisters[2221] := 16#0000;
   HoldingRegisters[2222] := 16#0000;
   HoldingRegisters[2223] := 16#0000;
   HoldingRegisters[2224] := 16#0000;
   HoldingRegisters[2225] := 16#0000;
   HoldingRegisters[2226] := 16#0000;
   HoldingRegisters[2227] := 16#0000;
   HoldingRegisters[2228] := 16#0000;
   HoldingRegisters[2229] := 16#0000;
   HoldingRegisters[2230] := 16#0000;
   HoldingRegisters[2231] := 16#0000;
   HoldingRegisters[2232] := 16#0000;
   HoldingRegisters[2233] := 16#0000;
   HoldingRegisters[2234] := 16#0000;
   HoldingRegisters[2235] := 16#0000;
   HoldingRegisters[2236] := 16#0000;
   HoldingRegisters[2237] := 16#0000;
   HoldingRegisters[2238] := 16#0000;
   HoldingRegisters[2239] := 16#0000;
   HoldingRegisters[2240] := 16#0000;
   HoldingRegisters[2241] := 16#0000;
   HoldingRegisters[2242] := 16#0000;
   HoldingRegisters[2243] := 16#0000;
   HoldingRegisters[2244] := 16#0000;
   HoldingRegisters[2245] := 16#0000;
   HoldingRegisters[2246] := 16#0000;
   HoldingRegisters[2247] := 16#0000;
   HoldingRegisters[2248] := 16#0000;
   HoldingRegisters[2249] := 16#0000;
   HoldingRegisters[2250] := 16#0000;
   HoldingRegisters[2251] := 16#0000;
   HoldingRegisters[2252] := 16#0000;
   HoldingRegisters[2253] := 16#0000;
   HoldingRegisters[2254] := 16#0000;
   HoldingRegisters[2255] := 16#0000;
   HoldingRegisters[2256] := 16#0000;
   HoldingRegisters[2257] := 16#0000;
   HoldingRegisters[2258] := 16#0000;
   HoldingRegisters[2259] := 16#0000;
   HoldingRegisters[2260] := 16#0000;
   HoldingRegisters[2261] := 16#0000;
   HoldingRegisters[2262] := 16#0000;
   HoldingRegisters[2263] := 16#0000;
   HoldingRegisters[2264] := 16#0000;
   HoldingRegisters[2265] := 16#0000;
   HoldingRegisters[2266] := 16#0000;
   HoldingRegisters[2267] := 16#0000;
   HoldingRegisters[2268] := 16#0000;
   HoldingRegisters[2269] := 16#0000;
   HoldingRegisters[2270] := 16#0000;
   HoldingRegisters[2271] := 16#0000;
   HoldingRegisters[2272] := 16#0000;
   HoldingRegisters[2273] := 16#0000;
   HoldingRegisters[2274] := 16#0000;
   HoldingRegisters[2275] := 16#0000;
   HoldingRegisters[2276] := 16#0000;
   HoldingRegisters[2277] := 16#0000;
   HoldingRegisters[2278] := 16#0000;
   HoldingRegisters[2279] := 16#0000;
   HoldingRegisters[2280] := 16#0000;
   HoldingRegisters[2281] := 16#0000;
   HoldingRegisters[2282] := 16#0000;
   HoldingRegisters[2283] := 16#0000;
   HoldingRegisters[2284] := 16#0000;
   HoldingRegisters[2285] := 16#0000;
   HoldingRegisters[2286] := 16#0000;
   HoldingRegisters[2287] := 16#0000;
   HoldingRegisters[2288] := 16#0000;
   HoldingRegisters[2289] := 16#0000;
   HoldingRegisters[2290] := 16#0000;
   HoldingRegisters[2291] := 16#0000;
   HoldingRegisters[2292] := 16#0000;
   HoldingRegisters[2293] := 16#0000;
   HoldingRegisters[2294] := 16#0000;
   HoldingRegisters[2295] := 16#0000;
   HoldingRegisters[2296] := 16#0000;
   HoldingRegisters[2297] := 16#0000;
   HoldingRegisters[2298] := 16#0000;
   HoldingRegisters[2299] := 16#0000;
   HoldingRegisters[2300] := 16#0000;
   HoldingRegisters[2301] := 16#0000;
   HoldingRegisters[2302] := 16#0000;
   HoldingRegisters[2303] := 16#0000;
   HoldingRegisters[2304] := 16#0000;
   HoldingRegisters[2305] := 16#0000;
   HoldingRegisters[2306] := 16#0000;
   HoldingRegisters[2307] := 16#0000;
   HoldingRegisters[2308] := 16#0000;
   HoldingRegisters[2309] := 16#0000;
   HoldingRegisters[2310] := 16#0000;
   HoldingRegisters[2311] := 16#0000;
   HoldingRegisters[2312] := 16#0000;
   HoldingRegisters[2313] := 16#0000;
   HoldingRegisters[2314] := 16#0000;
   HoldingRegisters[2315] := 16#0000;
   HoldingRegisters[2316] := 16#0000;
   HoldingRegisters[2317] := 16#0000;
   HoldingRegisters[2318] := 16#0000;
   HoldingRegisters[2319] := 16#0000;
   HoldingRegisters[2320] := 16#0000;
   HoldingRegisters[2321] := 16#0000;
   HoldingRegisters[2322] := 16#0000;
   HoldingRegisters[2323] := 16#0000;
   HoldingRegisters[2324] := 16#0000;
   HoldingRegisters[2325] := 16#0000;
   HoldingRegisters[2326] := 16#0000;
   HoldingRegisters[2327] := 16#0000;
   HoldingRegisters[2328] := 16#0000;
   HoldingRegisters[2329] := 16#0000;
   HoldingRegisters[2330] := 16#0000;
   HoldingRegisters[2331] := 16#0000;
   HoldingRegisters[2332] := 16#0000;
   HoldingRegisters[2333] := 16#0000;
   HoldingRegisters[2334] := 16#0000;
   HoldingRegisters[2335] := 16#0000;
   HoldingRegisters[2336] := 16#0000;
   HoldingRegisters[2337] := 16#0000;
   HoldingRegisters[2338] := 16#0000;
   HoldingRegisters[2339] := 16#0000;
   HoldingRegisters[2340] := 16#0000;
   HoldingRegisters[2341] := 16#0000;
   HoldingRegisters[2342] := 16#0000;
   HoldingRegisters[2343] := 16#0000;
   HoldingRegisters[2344] := 16#0000;
   HoldingRegisters[2345] := 16#0000;
   HoldingRegisters[2346] := 16#0000;
   HoldingRegisters[2347] := 16#0000;
   HoldingRegisters[2348] := 16#0000;
   HoldingRegisters[2349] := 16#0000;
   HoldingRegisters[2350] := 16#0000;
   HoldingRegisters[2351] := 16#0000;
   HoldingRegisters[2352] := 16#0000;
   HoldingRegisters[2353] := 16#0000;
   HoldingRegisters[2354] := 16#0000;
   HoldingRegisters[2355] := 16#0000;
   HoldingRegisters[2356] := 16#0000;
   HoldingRegisters[2357] := 16#0000;
   HoldingRegisters[2358] := 16#0000;
   HoldingRegisters[2359] := 16#0000;
   HoldingRegisters[2360] := 16#0000;
   HoldingRegisters[2361] := 16#0000;
   HoldingRegisters[2362] := 16#0000;
   HoldingRegisters[2363] := 16#0000;
   HoldingRegisters[2364] := 16#0000;
   HoldingRegisters[2365] := 16#0000;
   HoldingRegisters[2366] := 16#0000;
   HoldingRegisters[2367] := 16#0000;
   HoldingRegisters[2368] := 16#0000;
   HoldingRegisters[2369] := 16#0000;
   HoldingRegisters[2370] := 16#0000;
   HoldingRegisters[2371] := 16#0000;
   HoldingRegisters[2372] := 16#0000;
   HoldingRegisters[2373] := 16#0000;
   HoldingRegisters[2374] := 16#0000;
   HoldingRegisters[2375] := 16#0000;
   HoldingRegisters[2376] := 16#0000;
   HoldingRegisters[2377] := 16#0000;
   HoldingRegisters[2378] := 16#0000;
   HoldingRegisters[2379] := 16#0000;
   HoldingRegisters[2380] := 16#0000;
   HoldingRegisters[2381] := 16#0000;
   HoldingRegisters[2382] := 16#0000;
   HoldingRegisters[2383] := 16#0000;
   HoldingRegisters[2384] := 16#0000;
   HoldingRegisters[2385] := 16#0000;
   HoldingRegisters[2386] := 16#0000;
   HoldingRegisters[2387] := 16#0000;
   HoldingRegisters[2388] := 16#0000;
   HoldingRegisters[2389] := 16#0000;
   HoldingRegisters[2390] := 16#0000;
   HoldingRegisters[2391] := 16#0000;
   HoldingRegisters[2392] := 16#0000;
   HoldingRegisters[2393] := 16#0000;
   HoldingRegisters[2394] := 16#0000;
   HoldingRegisters[2395] := 16#0000;
   HoldingRegisters[2396] := 16#0000;
   HoldingRegisters[2397] := 16#0000;
   HoldingRegisters[2398] := 16#0000;
   HoldingRegisters[2399] := 16#0000;
   HoldingRegisters[2400] := 16#0000;
   HoldingRegisters[2401] := 16#0000;
   HoldingRegisters[2402] := 16#0000;
   HoldingRegisters[2403] := 16#0000;
   HoldingRegisters[2404] := 16#0000;
   HoldingRegisters[2405] := 16#0000;
   HoldingRegisters[2406] := 16#0000;
   HoldingRegisters[2407] := 16#0000;
   HoldingRegisters[2408] := 16#0000;
   HoldingRegisters[2409] := 16#0000;
   HoldingRegisters[2410] := 16#0000;
   HoldingRegisters[2411] := 16#0000;
   HoldingRegisters[2412] := 16#0000;
   HoldingRegisters[2413] := 16#0000;
   HoldingRegisters[2414] := 16#0000;
   HoldingRegisters[2415] := 16#0000;
   HoldingRegisters[2416] := 16#0000;
   HoldingRegisters[2417] := 16#0000;
   HoldingRegisters[2418] := 16#0000;
   HoldingRegisters[2419] := 16#0000;
   HoldingRegisters[2420] := 16#0000;
   HoldingRegisters[2421] := 16#0000;
   HoldingRegisters[2422] := 16#0000;
   HoldingRegisters[2423] := 16#0000;
   HoldingRegisters[2424] := 16#0000;
   HoldingRegisters[2425] := 16#0000;
   HoldingRegisters[2426] := 16#0000;
   HoldingRegisters[2427] := 16#0000;
   HoldingRegisters[2428] := 16#0000;
   HoldingRegisters[2429] := 16#0000;
   HoldingRegisters[2430] := 16#0000;
   HoldingRegisters[2431] := 16#0000;
   HoldingRegisters[2432] := 16#0000;
   HoldingRegisters[2433] := 16#0000;
   HoldingRegisters[2434] := 16#0000;
   HoldingRegisters[2435] := 16#0000;
   HoldingRegisters[2436] := 16#0000;
   HoldingRegisters[2437] := 16#0000;
   HoldingRegisters[2438] := 16#0000;
   HoldingRegisters[2439] := 16#0000;
   HoldingRegisters[2440] := 16#0000;
   HoldingRegisters[2441] := 16#0000;
   HoldingRegisters[2442] := 16#0000;
   HoldingRegisters[2443] := 16#0000;
   HoldingRegisters[2444] := 16#0000;
   HoldingRegisters[2445] := 16#0000;
   HoldingRegisters[2446] := 16#0000;
   HoldingRegisters[2447] := 16#0000;
   HoldingRegisters[2448] := 16#0000;
   HoldingRegisters[2449] := 16#0000;
   HoldingRegisters[2450] := 16#0000;
   HoldingRegisters[2451] := 16#0000;
   HoldingRegisters[2452] := 16#0000;
   HoldingRegisters[2453] := 16#0000;
   HoldingRegisters[2454] := 16#0000;
   HoldingRegisters[2455] := 16#0000;
   HoldingRegisters[2456] := 16#0000;
   HoldingRegisters[2457] := 16#0000;
   HoldingRegisters[2458] := 16#0000;
   HoldingRegisters[2459] := 16#0000;
   HoldingRegisters[2460] := 16#0000;
   HoldingRegisters[2461] := 16#0000;
   HoldingRegisters[2462] := 16#0000;
   HoldingRegisters[2463] := 16#0000;
   HoldingRegisters[2464] := 16#0000;
   HoldingRegisters[2465] := 16#0000;
   HoldingRegisters[2466] := 16#0000;
   HoldingRegisters[2467] := 16#0000;
   HoldingRegisters[2468] := 16#0000;
   HoldingRegisters[2469] := 16#0000;
   HoldingRegisters[2470] := 16#0000;
   HoldingRegisters[2471] := 16#0000;
   HoldingRegisters[2472] := 16#0000;
   HoldingRegisters[2473] := 16#0000;
   HoldingRegisters[2474] := 16#0000;
   HoldingRegisters[2475] := 16#0000;
   HoldingRegisters[2476] := 16#0000;
   HoldingRegisters[2477] := 16#0000;
   HoldingRegisters[2478] := 16#0000;
   HoldingRegisters[2479] := 16#0000;
   HoldingRegisters[2480] := 16#0000;
   HoldingRegisters[2481] := 16#0000;
   HoldingRegisters[2482] := 16#0000;
   HoldingRegisters[2483] := 16#0000;
   HoldingRegisters[2484] := 16#0000;
   HoldingRegisters[2485] := 16#0000;
   HoldingRegisters[2486] := 16#0000;
   HoldingRegisters[2487] := 16#0000;
   HoldingRegisters[2488] := 16#0000;
   HoldingRegisters[2489] := 16#0000;
   HoldingRegisters[2490] := 16#0000;
   HoldingRegisters[2491] := 16#0000;
   HoldingRegisters[2492] := 16#0000;
   HoldingRegisters[2493] := 16#0000;
   HoldingRegisters[2494] := 16#0000;
   HoldingRegisters[2495] := 16#0000;
   HoldingRegisters[2496] := 16#0000;
   HoldingRegisters[2497] := 16#0000;
   HoldingRegisters[2498] := 16#0000;
   HoldingRegisters[2499] := 16#0000;
   HoldingRegisters[2500] := 16#0000;
   HoldingRegisters[2501] := 16#0000;
   HoldingRegisters[2502] := 16#0000;
   HoldingRegisters[2503] := 16#0000;
   HoldingRegisters[2504] := 16#0000;
   HoldingRegisters[2505] := 16#0000;
   HoldingRegisters[2506] := 16#0000;
   HoldingRegisters[2507] := 16#0000;
   HoldingRegisters[2508] := 16#0000;
   HoldingRegisters[2509] := 16#0000;
   HoldingRegisters[2510] := 16#0000;
   HoldingRegisters[2511] := 16#0000;
   HoldingRegisters[2512] := 16#0000;
   HoldingRegisters[2513] := 16#0000;
   HoldingRegisters[2514] := 16#0000;
   HoldingRegisters[2515] := 16#0000;
   HoldingRegisters[2516] := 16#0000;
   HoldingRegisters[2517] := 16#0000;
   HoldingRegisters[2518] := 16#0000;
   HoldingRegisters[2519] := 16#0000;
   HoldingRegisters[2520] := 16#0000;
   HoldingRegisters[2521] := 16#0000;
   HoldingRegisters[2522] := 16#0000;
   HoldingRegisters[2523] := 16#0000;
   HoldingRegisters[2524] := 16#0000;
   HoldingRegisters[2525] := 16#0000;
   HoldingRegisters[2526] := 16#0000;
   HoldingRegisters[2527] := 16#0000;
   HoldingRegisters[2528] := 16#0000;
   HoldingRegisters[2529] := 16#0000;
   HoldingRegisters[2530] := 16#0000;
   HoldingRegisters[2531] := 16#0000;
   HoldingRegisters[2532] := 16#0000;
   HoldingRegisters[2533] := 16#0000;
   HoldingRegisters[2534] := 16#0000;
   HoldingRegisters[2535] := 16#0000;
   HoldingRegisters[2536] := 16#0000;
   HoldingRegisters[2537] := 16#0000;
   HoldingRegisters[2538] := 16#0000;
   HoldingRegisters[2539] := 16#0000;
   HoldingRegisters[2540] := 16#0000;
   HoldingRegisters[2541] := 16#0000;
   HoldingRegisters[2542] := 16#0000;
   HoldingRegisters[2543] := 16#0000;
   HoldingRegisters[2544] := 16#0000;
   HoldingRegisters[2545] := 16#0000;
   HoldingRegisters[2546] := 16#0000;
   HoldingRegisters[2547] := 16#0000;
   HoldingRegisters[2548] := 16#0000;
   HoldingRegisters[2549] := 16#0000;
   HoldingRegisters[2550] := 16#0000;
   HoldingRegisters[2551] := 16#0000;
   HoldingRegisters[2552] := 16#0000;
   HoldingRegisters[2553] := 16#0000;
   HoldingRegisters[2554] := 16#0000;
   HoldingRegisters[2555] := 16#0000;
   HoldingRegisters[2556] := 16#0000;
   HoldingRegisters[2557] := 16#0000;
   HoldingRegisters[2558] := 16#0000;
   HoldingRegisters[2559] := 16#0000;
   HoldingRegisters[2560] := 16#0000;
   HoldingRegisters[2561] := 16#0000;
   HoldingRegisters[2562] := 16#0000;
   HoldingRegisters[2563] := 16#0000;
   HoldingRegisters[2564] := 16#0000;
   HoldingRegisters[2565] := 16#0000;
   HoldingRegisters[2566] := 16#0000;
   HoldingRegisters[2567] := 16#0000;
   HoldingRegisters[2568] := 16#0000;
   HoldingRegisters[2569] := 16#0000;
   HoldingRegisters[2570] := 16#0000;
   HoldingRegisters[2571] := 16#0000;
   HoldingRegisters[2572] := 16#0000;
   HoldingRegisters[2573] := 16#0000;
   HoldingRegisters[2574] := 16#0000;
   HoldingRegisters[2575] := 16#0000;
   HoldingRegisters[2576] := 16#0000;
   HoldingRegisters[2577] := 16#0000;
   HoldingRegisters[2578] := 16#0000;
   HoldingRegisters[2579] := 16#0000;
   HoldingRegisters[2580] := 16#0000;
   HoldingRegisters[2581] := 16#0000;
   HoldingRegisters[2582] := 16#0000;
   HoldingRegisters[2583] := 16#0000;
   HoldingRegisters[2584] := 16#0000;
   HoldingRegisters[2585] := 16#0000;
   HoldingRegisters[2586] := 16#0000;
   HoldingRegisters[2587] := 16#0000;
   HoldingRegisters[2588] := 16#0000;
   HoldingRegisters[2589] := 16#0000;
   HoldingRegisters[2590] := 16#0000;
   HoldingRegisters[2591] := 16#0000;
   HoldingRegisters[2592] := 16#0000;
   HoldingRegisters[2593] := 16#0000;
   HoldingRegisters[2594] := 16#0000;
   HoldingRegisters[2595] := 16#0000;
   HoldingRegisters[2596] := 16#0000;
   HoldingRegisters[2597] := 16#0000;
   HoldingRegisters[2598] := 16#0000;
   HoldingRegisters[2599] := 16#0000;
   HoldingRegisters[2600] := 16#0000;
   HoldingRegisters[2601] := 16#0000;
   HoldingRegisters[2602] := 16#0000;
